(* IEC 61131-3 sources: SmartHomeNew/snapshots/2026-05-25 (part 4) *)

(* ---- FB_Water_Output_Reconciliation.st ---- *)
FUNCTION_BLOCK FB_Water_Output_Reconciliation
VAR_INPUT
    VI_Enable : BOOL;
    VI_System_Time_MS : UDINT;
END_VAR
VAR
    L_i : INT;
    L_Output : ST_Water_Output_Projection_State;
    L_Valve : ST_Water_Valve_Runtime_State;
    L_State : ST_Water_Output_Reconciliation_State;
    L_Any_Runtime_Mismatch : BOOL;
    L_Any_Confirmation_Mismatch : BOOL;
    L_Any_Conflict : BOOL;
END_VAR

IF NOT VI_Enable THEN
    GVL_Water_Output_Reconciliation.G_Runtime_Valid := FALSE;
    RETURN;
END_IF;

L_Any_Runtime_Mismatch := FALSE;
L_Any_Confirmation_Mismatch := FALSE;
L_Any_Conflict := FALSE;

FOR L_i := 1 TO GVL_CONSTANTS.C_MAX_FLOOD_SENSORS DO

    L_Output := GVL_Water_Output_Projection.G_Output_Projection_State[L_i];
    L_Valve := GVL_Water_Valve_Runtime.G_Valve_Runtime_State[L_i];

    // Reset all reconciliation fields per sensor to prevent state leakage across loop iterations.
    L_State.Runtime_Valid := FALSE;
    L_State.Runtime_System_Time_MS := 0;
    L_State.Valve_Group_Id := 0;
    L_State.Projection_Active := FALSE;
    L_State.Runtime_Output_Active := FALSE;
    L_State.Expected_Closed := FALSE;
    L_State.Confirmed_Closed := FALSE;
    L_State.Confirmation_Unknown := FALSE;
    L_State.Reconciliation_Healthy := FALSE;
    L_State.Projection_Runtime_Mismatch := FALSE;
    L_State.Projection_Confirmation_Mismatch := FALSE;
    L_State.Conflict_Detected := FALSE;
    L_State.Topology_Invalid := FALSE;
    L_State.Status_Code := 0;
    L_State.Status_Text := '';

    L_State.Runtime_Valid := TRUE;
    L_State.Runtime_System_Time_MS := VI_System_Time_MS;

    L_State.Valve_Group_Id := L_Output.Valve_Group_Id;
    L_State.Projection_Active := L_Output.Physical_Close_Project;
    L_State.Runtime_Output_Active := L_Valve.Physical_Output_Active;
    L_State.Expected_Closed := L_Output.Expected_Closed;
    L_State.Confirmed_Closed := L_Valve.Confirmed_Closed;
    L_State.Confirmation_Unknown := L_Valve.Confirmation_Unknown;

    IF L_Valve.Confirmation_Available THEN

        IF L_State.Projection_Active <> L_State.Runtime_Output_Active THEN
            L_State.Projection_Runtime_Mismatch := TRUE;
        END_IF;

        IF L_State.Expected_Closed
           AND NOT L_State.Confirmed_Closed THEN
            L_State.Projection_Confirmation_Mismatch := TRUE;
        END_IF;

    END_IF;

    IF L_Output.Projection_Allowed
       AND L_Output.Projection_Denied THEN
        L_State.Conflict_Detected := TRUE;
    END_IF;

    IF L_Output.Valve_Group_Id = 0 THEN
        L_State.Topology_Invalid := TRUE;
    END_IF;

    L_State.Reconciliation_Healthy :=
        NOT L_State.Projection_Runtime_Mismatch
        AND NOT L_State.Projection_Confirmation_Mismatch
        AND NOT L_State.Conflict_Detected
        AND NOT L_State.Topology_Invalid;

    IF L_State.Conflict_Detected THEN
        L_State.Status_Code := 3;
        L_State.Status_Text := 'Projection conflict detected';
    ELSIF L_State.Projection_Runtime_Mismatch THEN
        L_State.Status_Code := 2;
        L_State.Status_Text := 'Projection runtime mismatch';
        L_Any_Runtime_Mismatch := TRUE;
    ELSIF L_State.Projection_Confirmation_Mismatch THEN
        L_State.Status_Code := 1;
        L_State.Status_Text := 'Projection confirmation mismatch';
        L_Any_Confirmation_Mismatch := TRUE;
    ELSE
        L_State.Status_Code := 0;
        L_State.Status_Text := 'Reconciliation healthy';
    END_IF;

    IF L_State.Conflict_Detected THEN
        L_Any_Conflict := TRUE;
    END_IF;

    GVL_Water_Output_Reconciliation.G_Reconciliation_State[L_i] := L_State;
END_FOR;

GVL_Water_Output_Reconciliation.G_Any_Runtime_Mismatch := L_Any_Runtime_Mismatch;
GVL_Water_Output_Reconciliation.G_Any_Confirmation_Mismatch := L_Any_Confirmation_Mismatch;
GVL_Water_Output_Reconciliation.G_Any_Conflict_Detected := L_Any_Conflict;
GVL_Water_Output_Reconciliation.G_Runtime_Valid := TRUE;
GVL_Water_Output_Reconciliation.G_Last_Update_MS := VI_System_Time_MS;

IF L_Any_Conflict THEN
    GVL_Water_Output_Reconciliation.G_Status_Code := 3;
    GVL_Water_Output_Reconciliation.G_Status_Text := 'Water output reconciliation conflict';
ELSIF L_Any_Runtime_Mismatch THEN
    GVL_Water_Output_Reconciliation.G_Status_Code := 2;
    GVL_Water_Output_Reconciliation.G_Status_Text := 'Water output runtime mismatch';
ELSIF L_Any_Confirmation_Mismatch THEN
    GVL_Water_Output_Reconciliation.G_Status_Code := 1;
    GVL_Water_Output_Reconciliation.G_Status_Text := 'Water output confirmation mismatch';
ELSE
    GVL_Water_Output_Reconciliation.G_Status_Code := 0;
    GVL_Water_Output_Reconciliation.G_Status_Text := 'Water output reconciliation healthy';
END_IF;

END_FUNCTION_BLOCK

(* ---- MAIN.st ---- *)
PROGRAM MAIN
// ==============================================================================
// MAIN — deterministic PLC scan-cycle phase map.
// ==============================================================================
// Execution order is preserved by PRG_Main_Phase_* programs.
// No phase gating or controlled shedding is applied here yet.
// Compile/runtime validation must confirm that all referenced phase programs are
// linked by the PLC project export.
// ==============================================================================

PRG_Main_Phase_01_Bootstrap();
PRG_Main_Phase_02_Redundancy();
PRG_Main_Phase_03_Input_Safety_Command();
PRG_Main_Phase_04_Transport_Distributed();
PRG_Main_Phase_05_Domain_Output();
PRG_Main_Phase_06_PostOutput_Authority();
PRG_Main_Phase_07_Semantic_Governance();
PRG_Main_Phase_08_Diagnostics_HMI();

// >>> BULK_SYNC_ANCHOR: MAIN <<<
END_PROGRAM

(* ---- PRG_Access.st ---- *)
PROGRAM PRG_Access
VAR
    fbProjection : FB_Access_Output_Projection;

    fbPulseLock1Open : FB_Access_Pulse_Channel;
    fbPulseLock1Close : FB_Access_Pulse_Channel;
    fbPulseLock2Open : FB_Access_Pulse_Channel;
    fbPulseLock2Close : FB_Access_Pulse_Channel;
    fbPulseGateOpen : FB_Access_Pulse_Channel;
    fbPulseWicketOpen : FB_Access_Pulse_Channel;

    L_Mode : E_Safety_Mode;
    L_Now_MS : UDINT;
    L_Pulse_MS : UDINT;

    L_Distributed_Execute_Allowed : BOOL;
    L_Distributed_Access_Allowed : BOOL;

    L_Lock_1_Open : BOOL;
    L_Lock_1_Close : BOOL;
    L_Lock_2_Open : BOOL;
    L_Lock_2_Close : BOOL;
    L_Gate_Open : BOOL;
    L_Wicket_Open : BOOL;
END_VAR

L_Mode := GVL_SAFETY_SHUTDOWN.G_Safety_Mode;
L_Now_MS := GVL_STATUS.G_System_Time_MS;

GVL_ACCESS_RUNTIME.G_Runtime_Required := FALSE;
GVL_ACCESS_RUNTIME.G_Runtime_Executed := TRUE;
GVL_ACCESS_RUNTIME.G_Runtime_Idle_By_Design := FALSE;
GVL_ACCESS_RUNTIME.G_Runtime_Blocked_By_Distributed_Gates := FALSE;
GVL_ACCESS_RUNTIME.G_Any_Pulse_Active := FALSE;
GVL_ACCESS_RUNTIME.G_Last_Update_MS := L_Now_MS;

// Distributed runtime governance.
// FIRE/GAS emergency semantics remain authoritative.
L_Distributed_Execute_Allowed :=
    GVL_Distributed_Execution_Gates.G_Can_Execute;

L_Distributed_Access_Allowed :=
    GVL_Distributed_Execution_Gates.G_Can_Own_Projection;

IF (L_Mode <> FIRE)
   AND (L_Mode <> GAS)
   AND (
        NOT L_Distributed_Execute_Allowed
        OR NOT L_Distributed_Access_Allowed
       ) THEN

    // Clear all pulse channels before blocking projection to avoid stale pulse-active state.
    fbPulseLock1Open(VI_Command := FALSE, VI_Reset := TRUE, VI_Now_MS := L_Now_MS, VI_Pulse_MS := 100);
    fbPulseLock1Close(VI_Command := FALSE, VI_Reset := TRUE, VI_Now_MS := L_Now_MS, VI_Pulse_MS := 100);
    fbPulseLock2Open(VI_Command := FALSE, VI_Reset := TRUE, VI_Now_MS := L_Now_MS, VI_Pulse_MS := 100);
    fbPulseLock2Close(VI_Command := FALSE, VI_Reset := TRUE, VI_Now_MS := L_Now_MS, VI_Pulse_MS := 100);
    fbPulseGateOpen(VI_Command := FALSE, VI_Reset := TRUE, VI_Now_MS := L_Now_MS, VI_Pulse_MS := 100);
    fbPulseWicketOpen(VI_Command := FALSE, VI_Reset := TRUE, VI_Now_MS := L_Now_MS, VI_Pulse_MS := 100);

    fbProjection(
        VI_Lock_1_Open := FALSE,
        VI_Lock_1_Close := FALSE,
        VI_Lock_2_Open := FALSE,
        VI_Lock_2_Close := FALSE,
        VI_Gate_Open := FALSE,
        VI_Wicket_Open := FALSE
    );

    GVL_ACCESS_RUNTIME.G_Runtime_Blocked_By_Distributed_Gates := TRUE;
    GVL_ACCESS_RUNTIME.G_Any_Pulse_Active := FALSE;
    GVL_ACCESS_RUNTIME.G_Status_Code := 2;
    GVL_ACCESS_RUNTIME.G_Status_Text := 'Access runtime blocked by distributed gates';

    RETURN;
END_IF;

// Load pulse duration from config with safety clamp.
L_Pulse_MS := GVL_CONFIG.G_Access_Pulse_MS;
IF L_Pulse_MS < 100 THEN
    L_Pulse_MS := 100;
ELSIF L_Pulse_MS > 5000 THEN
    L_Pulse_MS := 5000;
END_IF;

L_Lock_1_Open := FALSE;
L_Lock_1_Close := FALSE;
L_Lock_2_Open := FALSE;
L_Lock_2_Close := FALSE;
L_Gate_Open := FALSE;
L_Wicket_Open := FALSE;

CASE L_Mode OF
    FIRE:
        // Fire evacuation access commands are authoritative and continuous.
        L_Lock_1_Open := GVL_COMMAND_SHADOW.G_Lock_1_Open;
        L_Lock_2_Open := GVL_COMMAND_SHADOW.G_Lock_2_Open;
        L_Gate_Open := GVL_COMMAND_SHADOW.G_Gate_Open;
        L_Wicket_Open := GVL_COMMAND_SHADOW.G_Wicket_Open;

        // Synchronize pulse channels with current command state and clear active pulses.
        fbPulseLock1Open(VI_Command := GVL_COMMAND_SHADOW.G_Lock_1_Open, VI_Reset := TRUE, VI_Now_MS := L_Now_MS, VI_Pulse_MS := L_Pulse_MS);
        fbPulseLock1Close(VI_Command := GVL_COMMAND_SHADOW.G_Lock_1_Close, VI_Reset := TRUE, VI_Now_MS := L_Now_MS, VI_Pulse_MS := L_Pulse_MS);
        fbPulseLock2Open(VI_Command := GVL_COMMAND_SHADOW.G_Lock_2_Open, VI_Reset := TRUE, VI_Now_MS := L_Now_MS, VI_Pulse_MS := L_Pulse_MS);
        fbPulseLock2Close(VI_Command := GVL_COMMAND_SHADOW.G_Lock_2_Close, VI_Reset := TRUE, VI_Now_MS := L_Now_MS, VI_Pulse_MS := L_Pulse_MS);
        fbPulseGateOpen(VI_Command := GVL_COMMAND_SHADOW.G_Gate_Open, VI_Reset := TRUE, VI_Now_MS := L_Now_MS, VI_Pulse_MS := L_Pulse_MS);
        fbPulseWicketOpen(VI_Command := GVL_COMMAND_SHADOW.G_Wicket_Open, VI_Reset := TRUE, VI_Now_MS := L_Now_MS, VI_Pulse_MS := L_Pulse_MS);

    GAS:
        // Gas mode uses direct gate opening plus limited pulsed pedestrian/lock release.
        L_Gate_Open := GVL_COMMAND_SHADOW.G_Gate_Open;

        fbPulseLock1Open(VI_Command := GVL_COMMAND_SHADOW.G_Lock_1_Open, VI_Reset := FALSE, VI_Now_MS := L_Now_MS, VI_Pulse_MS := L_Pulse_MS);
        fbPulseLock2Open(VI_Command := GVL_COMMAND_SHADOW.G_Lock_2_Open, VI_Reset := FALSE, VI_Now_MS := L_Now_MS, VI_Pulse_MS := L_Pulse_MS);
        fbPulseWicketOpen(VI_Command := GVL_COMMAND_SHADOW.G_Wicket_Open, VI_Reset := FALSE, VI_Now_MS := L_Now_MS, VI_Pulse_MS := L_Pulse_MS);

        fbPulseLock1Close(VI_Command := GVL_COMMAND_SHADOW.G_Lock_1_Close, VI_Reset := TRUE, VI_Now_MS := L_Now_MS, VI_Pulse_MS := L_Pulse_MS);
        fbPulseLock2Close(VI_Command := GVL_COMMAND_SHADOW.G_Lock_2_Close, VI_Reset := TRUE, VI_Now_MS := L_Now_MS, VI_Pulse_MS := L_Pulse_MS);
        fbPulseGateOpen(VI_Command := GVL_COMMAND_SHADOW.G_Gate_Open, VI_Reset := TRUE, VI_Now_MS := L_Now_MS, VI_Pulse_MS := L_Pulse_MS);

        L_Lock_1_Open := fbPulseLock1Open.VO_Output;
        L_Lock_2_Open := fbPulseLock2Open.VO_Output;
        L_Wicket_Open := fbPulseWicketOpen.VO_Output;

ELSE
        fbPulseLock1Open(VI_Command := GVL_COMMAND_SHADOW.G_Lock_1_Open, VI_Reset := FALSE, VI_Now_MS := L_Now_MS, VI_Pulse_MS := L_Pulse_MS);
        fbPulseLock1Close(VI_Command := GVL_COMMAND_SHADOW.G_Lock_1_Close, VI_Reset := FALSE, VI_Now_MS := L_Now_MS, VI_Pulse_MS := L_Pulse_MS);
        fbPulseLock2Open(VI_Command := GVL_COMMAND_SHADOW.G_Lock_2_Open, VI_Reset := FALSE, VI_Now_MS := L_Now_MS, VI_Pulse_MS := L_Pulse_MS);
        fbPulseLock2Close(VI_Command := GVL_COMMAND_SHADOW.G_Lock_2_Close, VI_Reset := FALSE, VI_Now_MS := L_Now_MS, VI_Pulse_MS := L_Pulse_MS);
        fbPulseGateOpen(VI_Command := GVL_COMMAND_SHADOW.G_Gate_Open, VI_Reset := FALSE, VI_Now_MS := L_Now_MS, VI_Pulse_MS := L_Pulse_MS);
        fbPulseWicketOpen(VI_Command := GVL_COMMAND_SHADOW.G_Wicket_Open, VI_Reset := FALSE, VI_Now_MS := L_Now_MS, VI_Pulse_MS := L_Pulse_MS);

        L_Lock_1_Open := fbPulseLock1Open.VO_Output;
        L_Lock_1_Close := fbPulseLock1Close.VO_Output;
        L_Lock_2_Open := fbPulseLock2Open.VO_Output;
        L_Lock_2_Close := fbPulseLock2Close.VO_Output;
        L_Gate_Open := fbPulseGateOpen.VO_Output;
        L_Wicket_Open := fbPulseWicketOpen.VO_Output;
END_CASE;

GVL_ACCESS_RUNTIME.G_Any_Pulse_Active :=
    fbPulseLock1Open.VO_Active
    OR fbPulseLock1Close.VO_Active
    OR fbPulseLock2Open.VO_Active
    OR fbPulseLock2Close.VO_Active
    OR fbPulseGateOpen.VO_Active
    OR fbPulseWicketOpen.VO_Active;

GVL_ACCESS_RUNTIME.G_Runtime_Required :=
    (L_Mode = FIRE)
    OR (L_Mode = GAS)
    OR GVL_COMMAND_SHADOW.G_Lock_1_Open
    OR GVL_COMMAND_SHADOW.G_Lock_1_Close
    OR GVL_COMMAND_SHADOW.G_Lock_2_Open
    OR GVL_COMMAND_SHADOW.G_Lock_2_Close
    OR GVL_COMMAND_SHADOW.G_Gate_Open
    OR GVL_COMMAND_SHADOW.G_Wicket_Open
    OR GVL_ACCESS_RUNTIME.G_Any_Pulse_Active;

GVL_ACCESS_RUNTIME.G_Runtime_Idle_By_Design :=
    NOT GVL_ACCESS_RUNTIME.G_Runtime_Required;

IF GVL_ACCESS_RUNTIME.G_Runtime_Idle_By_Design THEN
    GVL_ACCESS_RUNTIME.G_Status_Code := 0;
    GVL_ACCESS_RUNTIME.G_Status_Text := 'Access runtime idle by design';
ELSE
    GVL_ACCESS_RUNTIME.G_Status_Code := 1;
    GVL_ACCESS_RUNTIME.G_Status_Text := 'Access runtime active';
END_IF;

fbProjection(
    VI_Lock_1_Open := L_Lock_1_Open,
    VI_Lock_1_Close := L_Lock_1_Close,
    VI_Lock_2_Open := L_Lock_2_Open,
    VI_Lock_2_Close := L_Lock_2_Close,
    VI_Gate_Open := L_Gate_Open,
    VI_Wicket_Open := L_Wicket_Open
);

// >>> BULK_SYNC_ANCHOR: PRG_Access <<<
END_PROGRAM

(* ---- PRG_Authority_Lineage_Governor.st ---- *)
PROGRAM PRG_Authority_Lineage_Governor
VAR
    L_Now_MS : UDINT;
    L_Lineage_Valid : BOOL := TRUE;
    L_Error_Code : UDINT := 0;
    L_Error_Text : STRING(160) := '';
END_VAR

L_Now_MS := GVL_STATUS.G_System_Time_MS;
L_Lineage_Valid := TRUE;
L_Error_Code := 0;
L_Error_Text := '';

GVL_AUTHORITY_LINEAGE.Authority_Lineage_Valid := FALSE;
GVL_AUTHORITY_LINEAGE.Warm_Restart_Continuity_Valid := FALSE;
GVL_AUTHORITY_LINEAGE.HA_Resume_Continuity_Valid := FALSE;
GVL_AUTHORITY_LINEAGE.Retained_State_Integrity_Valid := FALSE;

IF GVL_AUTHORITY_LINEAGE.Authority_Replay_Suspected THEN
    L_Lineage_Valid := FALSE;
    L_Error_Code := 25000;
    L_Error_Text := 'Authority replay suspected';
END_IF;

IF L_Lineage_Valid AND GVL_AUTHORITY_LINEAGE.Retained_State_Skew_Detected THEN
    L_Lineage_Valid := FALSE;
    L_Error_Code := 25001;
    L_Error_Text := 'Retained state skew detected';
END_IF;

IF L_Lineage_Valid AND GVL_AUTHORITY_LINEAGE.Partial_Authority_Resurrection_Detected THEN
    L_Lineage_Valid := FALSE;
    L_Error_Code := 25002;
    L_Error_Text := 'Partial authority resurrection detected';
END_IF;

IF L_Lineage_Valid AND GVL_AUTHORITY_LINEAGE.Epoch_Lineage_Discontinuity_Detected THEN
    L_Lineage_Valid := FALSE;
    L_Error_Code := 25003;
    L_Error_Text := 'Epoch lineage discontinuity detected';
END_IF;

IF L_Lineage_Valid
AND (ULINT_TO_UDINT(GVL_PHYSICAL_AUTHORITY_EPOCH.Physical_Authority_Epoch) < GVL_AUTHORITY_LINEAGE.Last_Physical_Authority_Epoch) THEN
    GVL_AUTHORITY_LINEAGE.Authority_Replay_Suspected := TRUE;
    L_Lineage_Valid := FALSE;
    L_Error_Code := 25010;
    L_Error_Text := 'Physical authority epoch rollback detected';
END_IF;

IF L_Lineage_Valid
AND (ULINT_TO_UDINT(GVL_RUNTIME_EPOCH.Runtime_Epoch) < GVL_AUTHORITY_LINEAGE.Last_Runtime_Epoch) THEN
    GVL_AUTHORITY_LINEAGE.Retained_State_Skew_Detected := TRUE;
    L_Lineage_Valid := FALSE;
    L_Error_Code := 25011;
    L_Error_Text := 'Runtime epoch rollback detected';
END_IF;

IF L_Lineage_Valid
AND (ULINT_TO_UDINT(GVL_OUTPUT_EPOCH.Output_Publication_Epoch) < GVL_AUTHORITY_LINEAGE.Last_Output_Publication_Epoch) THEN
    GVL_AUTHORITY_LINEAGE.Partial_Authority_Resurrection_Detected := TRUE;
    L_Lineage_Valid := FALSE;
    L_Error_Code := 25012;
    L_Error_Text := 'Output publication epoch rollback detected';
END_IF;

IF L_Lineage_Valid THEN
    GVL_AUTHORITY_LINEAGE.Authority_Lineage_Valid := TRUE;
    GVL_AUTHORITY_LINEAGE.Warm_Restart_Continuity_Valid := TRUE;
    GVL_AUTHORITY_LINEAGE.HA_Resume_Continuity_Valid := TRUE;
    GVL_AUTHORITY_LINEAGE.Retained_State_Integrity_Valid := TRUE;

    GVL_AUTHORITY_LINEAGE.Authority_Lineage_Epoch := ULINT_TO_UDINT(GVL_PHYSICAL_AUTHORITY_EPOCH.Physical_Authority_Epoch);
    GVL_AUTHORITY_LINEAGE.Last_Physical_Authority_Epoch := ULINT_TO_UDINT(GVL_PHYSICAL_AUTHORITY_EPOCH.Physical_Authority_Epoch);
    GVL_AUTHORITY_LINEAGE.Last_Runtime_Epoch := ULINT_TO_UDINT(GVL_RUNTIME_EPOCH.Runtime_Epoch);
    GVL_AUTHORITY_LINEAGE.Last_Output_Publication_Epoch := ULINT_TO_UDINT(GVL_OUTPUT_EPOCH.Output_Publication_Epoch);
    GVL_AUTHORITY_LINEAGE.Authority_Lineage_Last_Update_MS := L_Now_MS;
    GVL_AUTHORITY_LINEAGE.Authority_Lineage_Last_Error_Code := 0;
    GVL_AUTHORITY_LINEAGE.Authority_Lineage_Last_Error_Text := '';
ELSE
    GVL_AUTHORITY_LINEAGE.Authority_Lineage_Valid := FALSE;
    GVL_AUTHORITY_LINEAGE.Authority_Lineage_Last_Error_Code := L_Error_Code;
    GVL_AUTHORITY_LINEAGE.Authority_Lineage_Last_Error_Text := L_Error_Text;
    GVL_AUTHORITY_LINEAGE.Authority_Lineage_Invalidation_Count := GVL_AUTHORITY_LINEAGE.Authority_Lineage_Invalidation_Count + 1;
END_IF;

END_PROGRAM

(* ---- PRG_Authority_Restoration_Governor.st ---- *)
PROGRAM PRG_Authority_Restoration_Governor
VAR
    L_Now_MS : UDINT;
    L_Restoration_Valid : BOOL := TRUE;
END_VAR

L_Now_MS := GVL_STATUS.G_System_Time_MS;
L_Restoration_Valid := TRUE;

GVL_AUTHORITY_RESTORATION.Authority_Restoration_Active := FALSE;
GVL_AUTHORITY_RESTORATION.Authority_Restoration_Allowed := FALSE;
GVL_AUTHORITY_RESTORATION.Authority_Restoration_Completed := FALSE;

GVL_AUTHORITY_RESTORATION.Snapshot_Restoration_Valid := FALSE;
GVL_AUTHORITY_RESTORATION.Consensus_Restoration_Valid := FALSE;
GVL_AUTHORITY_RESTORATION.Causality_Restoration_Valid := FALSE;
GVL_AUTHORITY_RESTORATION.Epoch_Restoration_Valid := FALSE;
GVL_AUTHORITY_RESTORATION.Lineage_Restoration_Valid := FALSE;

GVL_AUTHORITY_RESTORATION.Revocation_Clearance_Valid := FALSE;
GVL_AUTHORITY_RESTORATION.Stabilization_Window_Elapsed := FALSE;
GVL_AUTHORITY_RESTORATION.Reauthorization_Order_Valid := FALSE;

IF GVL_AUTHORITY_REVOCATION.Authority_Revocation_Active THEN
    L_Restoration_Valid := FALSE;
END_IF;

IF L_Restoration_Valid
AND (
    GVL_SAFETY_SHUTDOWN.G_Safety_Active
    OR GVL_SAFETY_RECOVERY.G_Recovery_Active
    OR (GVL_SAFETY_RECOVERY.G_Recovery_Phase <> IDLE)
) THEN
    L_Restoration_Valid := FALSE;
END_IF;

IF L_Restoration_Valid
AND NOT GVL_PHYSICAL_SNAPSHOT.Physical_Snapshot_Valid THEN
    L_Restoration_Valid := FALSE;
END_IF;

IF L_Restoration_Valid THEN
    GVL_AUTHORITY_RESTORATION.Snapshot_Restoration_Valid := TRUE;
END_IF;

IF L_Restoration_Valid
AND NOT GVL_SENSOR_CONSENSUS.Sensor_Consensus_Valid THEN
    L_Restoration_Valid := FALSE;
END_IF;

IF L_Restoration_Valid THEN
    GVL_AUTHORITY_RESTORATION.Consensus_Restoration_Valid := TRUE;
END_IF;

IF L_Restoration_Valid
AND NOT GVL_TELEMETRY.Command_Telemetry_Causality_Valid THEN
    L_Restoration_Valid := FALSE;
END_IF;

IF L_Restoration_Valid THEN
    GVL_AUTHORITY_RESTORATION.Causality_Restoration_Valid := TRUE;
END_IF;

IF L_Restoration_Valid
AND NOT GVL_PHYSICAL_AUTHORITY_EPOCH.Physical_Authority_Epoch_Valid THEN
    L_Restoration_Valid := FALSE;
END_IF;

IF L_Restoration_Valid THEN
    GVL_AUTHORITY_RESTORATION.Epoch_Restoration_Valid := TRUE;
END_IF;

IF L_Restoration_Valid
AND NOT GVL_AUTHORITY_LINEAGE.Authority_Lineage_Valid THEN
    L_Restoration_Valid := FALSE;
END_IF;

IF L_Restoration_Valid THEN
    GVL_AUTHORITY_RESTORATION.Lineage_Restoration_Valid := TRUE;
END_IF;

IF L_Restoration_Valid
AND GVL_AUTHORITY_REVOCATION.Quarantine_Fabric_Active THEN
    L_Restoration_Valid := FALSE;
END_IF;

IF L_Restoration_Valid THEN
    GVL_AUTHORITY_RESTORATION.Revocation_Clearance_Valid := TRUE;
END_IF;

IF L_Restoration_Valid
AND ((L_Now_MS - GVL_AUTHORITY_REVOCATION.Revocation_Last_Update_MS) < 5000) THEN
    L_Restoration_Valid := FALSE;
END_IF;

IF L_Restoration_Valid THEN
    GVL_AUTHORITY_RESTORATION.Stabilization_Window_Elapsed := TRUE;
END_IF;

IF L_Restoration_Valid THEN
    GVL_AUTHORITY_RESTORATION.Authority_Restoration_Active := TRUE;
    GVL_AUTHORITY_RESTORATION.Authority_Restoration_Allowed := TRUE;
    GVL_AUTHORITY_RESTORATION.Authority_Restoration_Completed := TRUE;
    GVL_AUTHORITY_RESTORATION.Reauthorization_Order_Valid := TRUE;
    GVL_AUTHORITY_RESTORATION.Restoration_Epoch :=
        GVL_PHYSICAL_AUTHORITY_EPOCH.Physical_Authority_Epoch;
    GVL_AUTHORITY_RESTORATION.Restoration_Last_Update_MS := L_Now_MS;
END_IF;

END_PROGRAM

(* ---- PRG_Away_Restore_Manager.st ---- *)
PROGRAM PRG_Away_Restore_Manager
VAR
    L_i : INT;
    L_Away_Active_Prev : BOOL := FALSE;
    L_Away_Level_Prev : BYTE := 0;
    L_Take_Snapshot : BOOL;
    L_Start_Restore : BOOL;
END_VAR

// Complete cleanup one cycle after publishing progress=1.0. This lets domain
// output managers consume the final restore state before snapshot invalidation.
IF GVL_AWAY_RESTORE.G_Restore_Finalize_Pending THEN
    GVL_AWAY_RESTORE.G_Restore_Active := FALSE;
    GVL_AWAY_RESTORE.G_Restore_Done := TRUE;
    GVL_AWAY_RESTORE.G_Snapshot_Valid := FALSE;
    GVL_AWAY_RESTORE.G_Restore_Finalize_Pending := FALSE;
    GVL_AWAY_RESTORE.G_Restore_Progress := 0.0;
END_IF;

L_Take_Snapshot :=
    GVL_POLICY.G_Away_Active AND
    (GVL_POLICY.G_Away_Level = 1) AND
    (NOT L_Away_Active_Prev);

IF L_Take_Snapshot THEN
    FOR L_i := 1 TO GVL_CONSTANTS.C_MAX_LIGHT_ZONES DO
        GVL_AWAY_RESTORE.G_Lighting_Levels[L_i] := GVL_STATE.G_Lighting_Levels[L_i];
    END_FOR;

    FOR L_i := 1 TO GVL_CONSTANTS.C_MAX_SOCKETS DO
        GVL_AWAY_RESTORE.G_Socket_States[L_i] := GVL_STATE.G_Socket_States[L_i];
    END_FOR;

    GVL_AWAY_RESTORE.G_Snapshot_Valid := TRUE;
    GVL_AWAY_RESTORE.G_Snapshot_Taken_MS := GVL_TIME_SERVICE.G_Now_MS;
    GVL_AWAY_RESTORE.G_Restore_Done := FALSE;
    GVL_AWAY_RESTORE.G_Restore_Finalize_Pending := FALSE;
END_IF;

L_Start_Restore :=
    GVL_POLICY.G_Away_Restore_Requested AND
    GVL_AWAY_RESTORE.G_Snapshot_Valid;

IF L_Start_Restore THEN
    GVL_AWAY_RESTORE.G_Restore_Active := TRUE;
    GVL_AWAY_RESTORE.G_Restore_Started_MS := GVL_TIME_SERVICE.G_Now_MS;
    GVL_AWAY_RESTORE.G_Restore_Done := FALSE;
    GVL_AWAY_RESTORE.G_Restore_Finalize_Pending := FALSE;
END_IF;

IF GVL_AWAY_RESTORE.G_Restore_Active THEN
    GVL_AWAY_RESTORE.G_Restore_Progress := GVL_POLICY.G_Away_Restore_Progress;

    IF NOT GVL_POLICY.G_Away_Restore_Active THEN
        GVL_AWAY_RESTORE.G_Restore_Progress := 1.0;
        GVL_AWAY_RESTORE.G_Restore_Finalize_Pending := TRUE;
    END_IF;
ELSE
    IF NOT GVL_AWAY_RESTORE.G_Restore_Done THEN
        GVL_AWAY_RESTORE.G_Restore_Progress := 0.0;
    END_IF;
END_IF;

L_Away_Active_Prev := GVL_POLICY.G_Away_Active;
L_Away_Level_Prev := GVL_POLICY.G_Away_Level;

END_PROGRAM

(* ---- PRG_Causal_Narrative_Engine.st ---- *)
PROGRAM PRG_Causal_Narrative_Engine
// PASSIVE CAUSAL NARRATIVE ENGINE
// HUMAN-READABLE SEMANTIC PROJECTION

GVL_CAUSAL_NARRATIVE_FABRIC.Narrative_Causality_Coherent :=
    GVL_TEMPORAL_CAUSALITY_CLOSURE_FABRIC.Temporal_Causality_Coherent;

GVL_CAUSAL_NARRATIVE_FABRIC.Narrative_Runtime_Alignment_Valid :=
    GVL_RUNTIME_TRANSITION_SYSTEM.Runtime_Transition_Legal;

IF GVL_RUNTIME_TRANSITION_SYSTEM.Illegal_Runtime_Transition_Observed THEN
    GVL_CAUSAL_NARRATIVE_FABRIC.Runtime_Narrative_Available := TRUE;
    GVL_CAUSAL_NARRATIVE_FABRIC.Runtime_Narrative_Code :=
        'transition legality violation observed';
END_IF;

IF GVL_RUNTIME_TRANSITION_SYSTEM.Recovery_Without_Lineage_Observed THEN
    GVL_CAUSAL_NARRATIVE_FABRIC.Recovery_Narrative_Available := TRUE;
    GVL_CAUSAL_NARRATIVE_FABRIC.Recovery_Narrative_Code :=
        'recovery blocked by lineage instability';
END_IF;

IF GVL_RUNTIME_TRANSITION_SYSTEM.Unsafe_Trust_Escalation_Observed THEN
    GVL_CAUSAL_NARRATIVE_FABRIC.Authority_Narrative_Available := TRUE;
    GVL_CAUSAL_NARRATIVE_FABRIC.Authority_Narrative_Code :=
        'unsafe trust escalation detected';
END_IF;

END_PROGRAM

(* ---- PRG_Causality_Reversal_Prevention_Governor.st ---- *)
PROGRAM PRG_Causality_Reversal_Prevention_Governor
IF GVL_HISTORICAL_ORDERING_INTEGRITY_FABRIC.Historical_Ordering_Integrity_Granted
AND NOT GVL_CAUSALITY_REVERSAL_PREVENTION_FABRIC.Causality_Reversal_Detected
AND NOT GVL_CAUSALITY_REVERSAL_PREVENTION_FABRIC.Resurrection_After_Revocation_Detected
AND NOT GVL_CAUSALITY_REVERSAL_PREVENTION_FABRIC.Unsafe_Temporal_Replay_Detected THEN

    GVL_CAUSALITY_REVERSAL_PREVENTION_FABRIC.Causality_Reversal_Prevention_Valid := TRUE;
    GVL_CAUSALITY_REVERSAL_PREVENTION_FABRIC.Causality_Reversal_Prevention_Granted := TRUE;
    GVL_CAUSALITY_REVERSAL_PREVENTION_FABRIC.Causality_Reversal_Prevented := TRUE;
    GVL_CAUSALITY_REVERSAL_PREVENTION_FABRIC.Authority_Ordering_Canonical := TRUE;
    GVL_CAUSALITY_REVERSAL_PREVENTION_FABRIC.Revocation_Resurrection_Boundary_Stable := TRUE;
END_IF;
END_PROGRAM

(* ---- PRG_Command_Arbitration_Phase_01_Reset_Role.st ---- *)
PROGRAM PRG_Command_Arbitration_Phase_01_Reset_Role
// Command arbitration phase 01: reset deterministic buffer and handle PLC role gates.
// Preserves old priority 1/2 early-exit semantics through buffer flags.

GVL_COMMAND_ARBITRATION_BUFFER.B_Mode := GVL_SAFETY_SHUTDOWN.G_Safety_Mode;
GVL_COMMAND_ARBITRATION_BUFFER.B_Safety_Active := FALSE;
GVL_COMMAND_ARBITRATION_BUFFER.B_User_Access_OK := FALSE;
GVL_COMMAND_ARBITRATION_BUFFER.B_Role_Conflict_Active := FALSE;
GVL_COMMAND_ARBITRATION_BUFFER.B_PLC_Inactive_Active := FALSE;

GVL_COMMAND_ARBITRATION_BUFFER.B_Gas_Valve_Close := FALSE;
GVL_COMMAND_ARBITRATION_BUFFER.B_Boiler_Stop := FALSE;
GVL_COMMAND_ARBITRATION_BUFFER.B_Supply_100_Req := FALSE;
GVL_COMMAND_ARBITRATION_BUFFER.B_Supply_80_Req := FALSE;
GVL_COMMAND_ARBITRATION_BUFFER.B_Vent_PV3_Boost := FALSE;
GVL_COMMAND_ARBITRATION_BUFFER.B_Exhaust_100_Req := FALSE;
GVL_COMMAND_ARBITRATION_BUFFER.B_Vent_Stop := FALSE;
GVL_COMMAND_ARBITRATION_BUFFER.B_Vent_Block := FALSE;
GVL_COMMAND_ARBITRATION_BUFFER.B_Vent_Smoke_Exhaust := FALSE;

GVL_COMMAND_ARBITRATION_BUFFER.B_Heating_Block := FALSE;
GVL_COMMAND_ARBITRATION_BUFFER.B_Heating_Emergency_Stop := FALSE;
GVL_COMMAND_ARBITRATION_BUFFER.B_Heating_Gas_Safety_Stop := FALSE;

GVL_COMMAND_ARBITRATION_BUFFER.B_Water_Block := FALSE;
GVL_COMMAND_ARBITRATION_BUFFER.B_Water_Emergency_Stop := FALSE;
GVL_COMMAND_ARBITRATION_BUFFER.B_Close_Valve_35 := FALSE;
GVL_COMMAND_ARBITRATION_BUFFER.B_Close_Valve_36 := FALSE;

GVL_COMMAND_ARBITRATION_BUFFER.B_Lock_1_Open := FALSE;
GVL_COMMAND_ARBITRATION_BUFFER.B_Lock_1_Close := FALSE;
GVL_COMMAND_ARBITRATION_BUFFER.B_Lock_2_Open := FALSE;
GVL_COMMAND_ARBITRATION_BUFFER.B_Lock_2_Close := FALSE;
GVL_COMMAND_ARBITRATION_BUFFER.B_Gate_Open := FALSE;
GVL_COMMAND_ARBITRATION_BUFFER.B_Wicket_Open := FALSE;

IF GVL_STATUS.G_Is_Active_PLC AND GVL_STATUS.G_Other_PLC_Is_Active THEN
    GVL_HEALTH_BRIDGE.G_Role_Conflict_Error := TRUE;
    GVL_COMMAND_ARBITRATION_BUFFER.B_Role_Conflict_Active := TRUE;

    GVL_COMMAND_ARBITRATION_BUFFER.B_Gas_Valve_Close := TRUE;
    GVL_COMMAND_ARBITRATION_BUFFER.B_Boiler_Stop := TRUE;
    GVL_COMMAND_ARBITRATION_BUFFER.B_Vent_Stop := TRUE;
    GVL_COMMAND_ARBITRATION_BUFFER.B_Vent_Block := TRUE;

    GVL_COMMAND_ARBITRATION_BUFFER.B_Heating_Block := TRUE;
    GVL_COMMAND_ARBITRATION_BUFFER.B_Heating_Emergency_Stop := TRUE;
    GVL_COMMAND_ARBITRATION_BUFFER.B_Heating_Gas_Safety_Stop := TRUE;

    GVL_COMMAND_ARBITRATION_BUFFER.B_Water_Block := TRUE;
    GVL_COMMAND_ARBITRATION_BUFFER.B_Water_Emergency_Stop := TRUE;
    GVL_COMMAND_ARBITRATION_BUFFER.B_Close_Valve_35 := TRUE;
    GVL_COMMAND_ARBITRATION_BUFFER.B_Close_Valve_36 := TRUE;

ELSIF NOT GVL_STATUS.G_Is_Active_PLC THEN
    GVL_COMMAND_ARBITRATION_BUFFER.B_PLC_Inactive_Active := TRUE;

    GVL_COMMAND_ARBITRATION_BUFFER.B_Gas_Valve_Close := GVL_COMMAND_POLICY_CONFIG.G_PLC_Inactive_Close_Gas;
    GVL_COMMAND_ARBITRATION_BUFFER.B_Boiler_Stop := GVL_COMMAND_POLICY_CONFIG.G_PLC_Inactive_Stop_Boiler;
    GVL_COMMAND_ARBITRATION_BUFFER.B_Vent_Stop := GVL_COMMAND_POLICY_CONFIG.G_PLC_Inactive_Stop_Vent;
    GVL_COMMAND_ARBITRATION_BUFFER.B_Vent_Block := FALSE;

    GVL_COMMAND_ARBITRATION_BUFFER.B_Heating_Block := GVL_COMMAND_POLICY_CONFIG.G_PLC_Inactive_Block_Heating;
    GVL_COMMAND_ARBITRATION_BUFFER.B_Heating_Emergency_Stop := FALSE;
    GVL_COMMAND_ARBITRATION_BUFFER.B_Heating_Gas_Safety_Stop := FALSE;

    GVL_COMMAND_ARBITRATION_BUFFER.B_Water_Block := GVL_COMMAND_POLICY_CONFIG.G_PLC_Inactive_Block_Water;
    GVL_COMMAND_ARBITRATION_BUFFER.B_Water_Emergency_Stop := FALSE;
    GVL_COMMAND_ARBITRATION_BUFFER.B_Close_Valve_35 := FALSE;
    GVL_COMMAND_ARBITRATION_BUFFER.B_Close_Valve_36 := FALSE;
END_IF;

// >>> BULK_SYNC_ANCHOR: PRG_Command_Arbitration_Phase_01_Reset_Role <<<
END_PROGRAM

(* ---- PRG_Convergence_Governor.st ---- *)
PROGRAM PRG_Convergence_Governor
VAR
    L_Now_MS : UDINT;
    L_Healthy : BOOL := TRUE;
    L_Error_Code : UDINT := 0;
    L_Error_Text : STRING(160) := '';

    L_Recent_Invalidation : BOOL;
    L_Epoch_Advancement_Healthy : BOOL;
END_VAR

L_Now_MS := GVL_STATUS.G_System_Time_MS;
L_Healthy := TRUE;
L_Error_Code := 0;
L_Error_Text := '';

GVL_CONVERGENCE.Convergence_Runtime_Barrier_OK :=
    GVL_RUNTIME_EPOCH.Runtime_Runtime_Barrier_OK
    AND GVL_RUNTIME_EPOCH.Runtime_IO_Publication_Allowed;

GVL_CONVERGENCE.Convergence_Runtime_Snapshot_OK :=
    GVL_RUNTIME_SNAPSHOT.Snapshot_Frozen
    AND GVL_RUNTIME_SNAPSHOT.Snapshot_Publication_Allowed
    AND GVL_RUNTIME_SNAPSHOT.Snapshot_Copy_Valid
    AND GVL_RUNTIME_SNAPSHOT.Snapshot_Isolation_Valid
    AND GVL_RUNTIME_SNAPSHOT.Snapshot_Runtime_Authority_Valid
    AND NOT GVL_RUNTIME_SNAPSHOT.Snapshot_Mutation_Detected;

GVL_CONVERGENCE.Convergence_Distributed_Snapshot_OK :=
    GVL_DISTRIBUTED_SNAPSHOT.Distributed_Publication_Reconciled
    AND GVL_DISTRIBUTED_SNAPSHOT.Distributed_Publication_Freeze_Valid
    AND GVL_DISTRIBUTED_SNAPSHOT.Distributed_Snapshot_Consistent;

GVL_CONVERGENCE.Convergence_Distributed_Commit_OK :=
    GVL_DISTRIBUTED_COMMIT.Distributed_Commit_Valid
    AND GVL_DISTRIBUTED_COMMIT.Publication_Prepare_Valid
    AND GVL_DISTRIBUTED_COMMIT.Publication_Commit_Confirmed
    AND NOT GVL_DISTRIBUTED_COMMIT.Peer_Commit_Mismatch
    AND NOT GVL_DISTRIBUTED_COMMIT.Commit_Lease_Expired;

GVL_CONVERGENCE.Convergence_Semantic_Progress_OK :=
    GVL_SEMANTIC_PROGRESS.Semantic_Forward_Progress_Valid
    AND GVL_SEMANTIC_PROGRESS.Semantic_Execution_Continuity_OK
    AND NOT GVL_SEMANTIC_PROGRESS.Semantic_Stagnation_Detected
    AND NOT GVL_SEMANTIC_PROGRESS.Semantic_Replay_Suspected
    AND NOT GVL_SEMANTIC_PROGRESS.Semantic_Livelock_Suspected
    AND NOT GVL_SEMANTIC_PROGRESS.Semantic_Deadlock_Suspected
    AND NOT GVL_SEMANTIC_PROGRESS.Semantic_Progress_Lease_Expired
    AND NOT GVL_SEMANTIC_PROGRESS.Semantic_Progress_Quarantine_Active;

GVL_CONVERGENCE.Convergence_Output_Freshness_OK :=
    GVL_RUNTIME_EPOCH.Runtime_Runtime_Barrier_OK
    AND GVL_RUNTIME_EPOCH.Runtime_IO_Publication_Allowed
    AND GVL_RUNTIME_SNAPSHOT.Snapshot_Frozen
    AND GVL_RUNTIME_SNAPSHOT.Snapshot_Publication_Allowed
    AND GVL_RUNTIME_SNAPSHOT.Snapshot_Copy_Valid
    AND GVL_RUNTIME_SNAPSHOT.Snapshot_Isolation_Valid
    AND NOT GVL_RUNTIME_SNAPSHOT.Snapshot_Mutation_Detected
    AND GVL_DISTRIBUTED_SNAPSHOT.Distributed_Publication_Reconciled
    AND GVL_DISTRIBUTED_SNAPSHOT.Distributed_Publication_Freeze_Valid
    AND GVL_DISTRIBUTED_SNAPSHOT.Distributed_Snapshot_Consistent
    AND GVL_DISTRIBUTED_COMMIT.Distributed_Commit_Valid
    AND GVL_DISTRIBUTED_COMMIT.Publication_Prepare_Valid
    AND GVL_DISTRIBUTED_COMMIT.Publication_Commit_Confirmed
    AND NOT GVL_DISTRIBUTED_COMMIT.Peer_Commit_Mismatch
    AND NOT GVL_DISTRIBUTED_COMMIT.Commit_Lease_Expired
    AND GVL_OUTPUT_EPOCH.Output_Publication_Valid
    AND GVL_OUTPUT_EPOCH.Output_Runtime_Epoch_Valid
    AND NOT GVL_OUTPUT_EPOCH.Output_Lease_Expired
    AND NOT GVL_OUTPUT_EPOCH.Output_Forced_Safe_Decay
    AND GVL_COMMAND_VERIFY.PreOutput_Barrier_OK
    AND NOT GVL_COMMAND_VERIFY.PreOutput_Block_IO;

// Epoch advancement freshness.
L_Epoch_Advancement_Healthy :=
    (GVL_SEMANTIC_PROGRESS.Semantic_Runtime_Barrier_Epoch -
     GVL_SEMANTIC_PROGRESS.Semantic_Last_Runtime_Barrier_Epoch) <= 2
    AND
    (GVL_SEMANTIC_PROGRESS.Semantic_Distributed_Commit_Epoch -
     GVL_SEMANTIC_PROGRESS.Semantic_Last_Distributed_Commit_Epoch) <= 2
    AND
    (GVL_SEMANTIC_PROGRESS.Semantic_Output_Publication_Epoch -
     GVL_SEMANTIC_PROGRESS.Semantic_Last_Output_Publication_Epoch) <= 2;

// Oscillation damping window.
L_Recent_Invalidation :=
    (L_Now_MS - GVL_CONVERGENCE.Convergence_Last_Invalidation_MS) < 30000;

IF NOT GVL_CONVERGENCE.Convergence_Runtime_Barrier_OK THEN
    L_Healthy := FALSE;
    L_Error_Code := 18000;
    L_Error_Text := 'Runtime barrier convergence invalid';
END_IF;

IF L_Healthy AND NOT GVL_CONVERGENCE.Convergence_Runtime_Snapshot_OK THEN
    L_Healthy := FALSE;
    L_Error_Code := 18001;
    L_Error_Text := 'Runtime snapshot convergence invalid';
END_IF;

IF L_Healthy AND NOT GVL_CONVERGENCE.Convergence_Distributed_Snapshot_OK THEN
    L_Healthy := FALSE;
    L_Error_Code := 18002;
    L_Error_Text := 'Distributed snapshot convergence invalid';
END_IF;

IF L_Healthy AND NOT GVL_CONVERGENCE.Convergence_Distributed_Commit_OK THEN
    L_Healthy := FALSE;
    L_Error_Code := 18003;
    L_Error_Text := 'Distributed commit convergence invalid';
END_IF;

IF L_Healthy AND NOT GVL_CONVERGENCE.Convergence_Semantic_Progress_OK THEN
    L_Healthy := FALSE;
    L_Error_Code := 18004;
    L_Error_Text := 'Semantic progress convergence invalid';
END_IF;

IF L_Healthy AND NOT GVL_CONVERGENCE.Convergence_Output_Freshness_OK THEN
    L_Healthy := FALSE;
    L_Error_Code := 18005;
    L_Error_Text := 'Output freshness convergence invalid';
END_IF;

IF L_Healthy AND NOT L_Epoch_Advancement_Healthy THEN
    L_Healthy := FALSE;
    L_Error_Code := 18006;
    L_Error_Text := 'Epoch advancement freshness invalid';
END_IF;

IF L_Healthy AND L_Recent_Invalidation THEN
    L_Healthy := FALSE;
    L_Error_Code := 18007;
    L_Error_Text := 'Convergence oscillation damping active';
END_IF;

IF L_Healthy THEN
    GVL_CONVERGENCE.Convergence_Healthy_Observed := TRUE;

    GVL_CONVERGENCE.Recovery_Stable_Cycle_Count :=
        GVL_CONVERGENCE.Recovery_Stable_Cycle_Count + 1;

    IF GVL_CONVERGENCE.Convergence_Last_Healthy_MS = 0 THEN
        GVL_CONVERGENCE.Convergence_Last_Healthy_MS := L_Now_MS;
    END_IF;

    GVL_CONVERGENCE.Recovery_Stable_Time_MS :=
        L_Now_MS - GVL_CONVERGENCE.Convergence_Last_Healthy_MS;

    IF (GVL_CONVERGENCE.Recovery_Stable_Cycle_Count >= GVL_CONVERGENCE.Convergence_Min_Stable_Cycles)
    AND (GVL_CONVERGENCE.Recovery_Stable_Time_MS >= GVL_CONVERGENCE.Convergence_Min_Stable_Time_MS)
    THEN
        GVL_CONVERGENCE.Convergence_Lease_OK := TRUE;
        GVL_CONVERGENCE.Convergence_Release_Allowed := TRUE;
    ELSE
        GVL_CONVERGENCE.Convergence_Lease_OK := FALSE;
        GVL_CONVERGENCE.Convergence_Release_Allowed := FALSE;
    END_IF;

    GVL_CONVERGENCE.Convergence_Last_Error_Code := 0;
    GVL_CONVERGENCE.Convergence_Last_Error_Text := '';
ELSE
    GVL_CONVERGENCE.Convergence_Healthy_Observed := FALSE;

    GVL_CONVERGENCE.Recovery_Stable_Cycle_Count := 0;
    GVL_CONVERGENCE.Recovery_Stable_Time_MS := 0;

    GVL_CONVERGENCE.Convergence_Lease_OK := FALSE;
    GVL_CONVERGENCE.Convergence_Release_Allowed := FALSE;

    GVL_CONVERGENCE.Convergence_Last_Healthy_MS := 0;
    GVL_CONVERGENCE.Convergence_Last_Invalidation_MS := L_Now_MS;

    GVL_CONVERGENCE.Convergence_Invalidation_Count :=
        GVL_CONVERGENCE.Convergence_Invalidation_Count + 1;

    // Oscillation quarantine.
    IF GVL_CONVERGENCE.Convergence_Invalidation_Count > 5 THEN
        GVL_CONVERGENCE.Convergence_Oscillation_Quarantine_Active := TRUE;
    END_IF;

    GVL_CONVERGENCE.Convergence_Last_Error_Code := L_Error_Code;
    GVL_CONVERGENCE.Convergence_Last_Error_Text := L_Error_Text;
END_IF;

END_PROGRAM

(* ---- PRG_CrossDomain_FailSafe_Closure_Governor.st ---- *)
PROGRAM PRG_CrossDomain_FailSafe_Closure_Governor
VAR
    L_Now_MS : UDINT;
    L_Valid : BOOL := TRUE;
END_VAR

L_Now_MS := GVL_STATUS.G_System_Time_MS;

GVL_CROSSDOMAIN_FAILSAFE_CLOSURE_FABRIC.CrossDomain_FailSafe_Closure_Valid := FALSE;
GVL_CROSSDOMAIN_FAILSAFE_CLOSURE_FABRIC.CrossDomain_FailSafe_Closure_Granted := FALSE;
GVL_CROSSDOMAIN_FAILSAFE_CLOSURE_FABRIC.CrossDomain_FailSafe_Closure_Quarantine_Active := TRUE;

IF NOT GVL_PHYSICAL_SAFESTATE_LATTICE_FABRIC.Physical_SafeState_Lattice_Granted THEN
    L_Valid := FALSE;
END_IF;

IF GVL_CROSSDOMAIN_FAILSAFE_CLOSURE_FABRIC.CrossDomain_FailSafe_Conflict_Detected
OR GVL_CROSSDOMAIN_FAILSAFE_CLOSURE_FABRIC.Unsafe_Recovery_Topology_Detected
OR GVL_CROSSDOMAIN_FAILSAFE_CLOSURE_FABRIC.CrossDomain_Recovery_Race_Detected
OR GVL_CROSSDOMAIN_FAILSAFE_CLOSURE_FABRIC.Distributed_SafeState_Fork_Detected
OR GVL_CROSSDOMAIN_FAILSAFE_CLOSURE_FABRIC.PowerDomain_Unsafe_Reactivation_Detected
OR GVL_CROSSDOMAIN_FAILSAFE_CLOSURE_FABRIC.MultiDomain_Recovery_Deadlock_Detected THEN
    L_Valid := FALSE;
END_IF;

IF L_Valid THEN
    GVL_CROSSDOMAIN_FAILSAFE_CLOSURE_FABRIC.CrossDomain_FailSafe_Closure_Valid := TRUE;
    GVL_CROSSDOMAIN_FAILSAFE_CLOSURE_FABRIC.CrossDomain_FailSafe_Closure_Granted := TRUE;
    GVL_CROSSDOMAIN_FAILSAFE_CLOSURE_FABRIC.CrossDomain_FailSafe_Closure_Quarantine_Active := FALSE;

    GVL_CROSSDOMAIN_FAILSAFE_CLOSURE_FABRIC.CrossDomain_SafeState_Compatibility_Valid := TRUE;
    GVL_CROSSDOMAIN_FAILSAFE_CLOSURE_FABRIC.FailSafe_Topology_Closure_Canonical := TRUE;
    GVL_CROSSDOMAIN_FAILSAFE_CLOSURE_FABRIC.MultiDomain_SafeTransition_Stable := TRUE;
    GVL_CROSSDOMAIN_FAILSAFE_CLOSURE_FABRIC.SafeState_Recovery_Ordering_Bounded := TRUE;
    GVL_CROSSDOMAIN_FAILSAFE_CLOSURE_FABRIC.Physical_Domain_Isolation_Coherent := TRUE;

    GVL_CROSSDOMAIN_FAILSAFE_CLOSURE_FABRIC.CrossDomain_FailSafe_Closure_Epoch :=
        GVL_PHYSICAL_SAFESTATE_LATTICE_FABRIC.Physical_SafeState_Lattice_Epoch;

    GVL_CROSSDOMAIN_FAILSAFE_CLOSURE_FABRIC.CrossDomain_FailSafe_Closure_Epoch_Coherent := TRUE;
    GVL_CROSSDOMAIN_FAILSAFE_CLOSURE_FABRIC.CrossDomain_FailSafe_Closure_Last_Update_MS := L_Now_MS;
    GVL_CROSSDOMAIN_FAILSAFE_CLOSURE_FABRIC.CrossDomain_FailSafe_Closure_Lease_Expired := FALSE;
END_IF;

END_PROGRAM

(* ---- PRG_Debug_View.st ---- *)
PROGRAM PRG_Debug_View
VAR
    L_i : INT;
    L_MaxWeight : REAL;
    L_MinWeight : REAL;
    L_Weight : REAL;
    L_Index : INT;
END_VAR

GVL_DEBUG_VIEW.D_Current_Time_MS := GVL_TIME_SERVICE.G_Now_MS;

GVL_DEBUG_VIEW.D_Safety_Mode := GVL_SAFETY_SHUTDOWN.G_Safety_Mode;
GVL_DEBUG_VIEW.D_Safety_Active := (GVL_SAFETY_SHUTDOWN.G_Safety_Mode <> NORMAL);
GVL_DEBUG_VIEW.D_Recovery_Phase := GVL_SAFETY_RECOVERY.G_Recovery_Phase;
GVL_DEBUG_VIEW.D_Recovery_Active := GVL_SAFETY_RECOVERY.G_Recovery_Active;
GVL_DEBUG_VIEW.D_Recovery_Exit_Allowed := GVL_SAFETY_RECOVERY.G_Recovery_Exit_Allowed;
GVL_DEBUG_VIEW.D_Authority_Revocation_Active := GVL_AUTHORITY_REVOCATION.Authority_Revocation_Active;
GVL_DEBUG_VIEW.D_Authority_Restoration_Allowed := GVL_AUTHORITY_RESTORATION.Authority_Restoration_Allowed;
GVL_DEBUG_VIEW.D_Authority_Restoration_Completed := GVL_AUTHORITY_RESTORATION.Authority_Restoration_Completed;

GVL_DEBUG_VIEW.D_Current_Scenario := GVL_INTENT_BEHAVIOR.I_Selected_Scenario_Text;
GVL_DEBUG_VIEW.D_Behavior_Reason := GVL_INTENT_BEHAVIOR.I_Reason_Text;

GVL_DEBUG_VIEW.D_Score_Night := GVL_INTENT_BEHAVIOR.I_Score_Night;
GVL_DEBUG_VIEW.D_Score_Preheat := GVL_INTENT_BEHAVIOR.I_Score_Preheat;
GVL_DEBUG_VIEW.D_Score_VentBoost := GVL_INTENT_BEHAVIOR.I_Score_Vent_Boost;
GVL_DEBUG_VIEW.D_Score_AccessSecure := GVL_INTENT_BEHAVIOR.I_Score_Access_Secure;

GVL_DEBUG_VIEW.D_Intent_Night := GVL_INTENT_BEHAVIOR.I_Request_Night_Mode;
GVL_DEBUG_VIEW.D_Intent_Comfort := GVL_INTENT_BEHAVIOR.I_Request_Comfort_Mode;
GVL_DEBUG_VIEW.D_Intent_VentBoost := GVL_INTENT_BEHAVIOR.I_Request_Ventilation_Boost;
GVL_DEBUG_VIEW.D_Intent_AccessSecure := GVL_INTENT_BEHAVIOR.I_Request_Access_Secure_Mode;

GVL_DEBUG_VIEW.D_Heating_Block := GVL_COMMAND_SHADOW.G_Heating_Block;
GVL_DEBUG_VIEW.D_Vent_Stop := GVL_COMMAND_SHADOW.G_Vent_Stop;
GVL_DEBUG_VIEW.D_Water_Block := GVL_COMMAND_SHADOW.G_Water_Block;
GVL_DEBUG_VIEW.D_Access_Open_Active := GVL_COMMAND_SHADOW.G_Gate_Open OR GVL_COMMAND_SHADOW.G_Wicket_Open;

GVL_DEBUG_VIEW.D_Global_Reason := GVL_EXPLAINABILITY.G_Last_Global_Reason_Text;
GVL_DEBUG_VIEW.D_Behavior_Why_Active := GVL_EXPLAINABILITY.G_Behavior_Why_Active;
GVL_DEBUG_VIEW.D_Heating_Why_Blocked := GVL_EXPLAINABILITY.G_Heating_Why_Blocked;
GVL_DEBUG_VIEW.D_Vent_Why_Stopped := GVL_EXPLAINABILITY.G_Vent_Why_Stopped;
GVL_DEBUG_VIEW.D_Water_Why_Closed := GVL_EXPLAINABILITY.G_Water_Why_Closed;
GVL_DEBUG_VIEW.D_Access_Why_Opened := GVL_EXPLAINABILITY.G_Access_Why_Opened;

// MAIN PHASE FEEDBACK SUMMARY -> DEBUG VIEW
GVL_DEBUG_VIEW.D_Main_Phase_Current := GVL_MAIN_PHASE_FEEDBACK.G_Current_Phase;
GVL_DEBUG_VIEW.D_Main_Phase_Critical_Executed := GVL_MAIN_PHASE_FEEDBACK.G_Critical_Path_Executed;
GVL_DEBUG_VIEW.D_Main_Phase_Critical_Valid := GVL_MAIN_PHASE_FEEDBACK.G_Critical_Path_Valid;
GVL_DEBUG_VIEW.D_Main_Phase_Observability_Executed := GVL_MAIN_PHASE_FEEDBACK.G_Observability_Path_Executed;
GVL_DEBUG_VIEW.D_Main_Phase_Observability_Valid := GVL_MAIN_PHASE_FEEDBACK.G_Observability_Path_Valid;
GVL_DEBUG_VIEW.D_Main_Phase_Any_Invalid := GVL_MAIN_PHASE_FEEDBACK.G_Any_Phase_Invalid;
GVL_DEBUG_VIEW.D_Main_Phase_Any_Skipped_By_Design := GVL_MAIN_PHASE_FEEDBACK.G_Any_Phase_Skipped_By_Design;
GVL_DEBUG_VIEW.D_Main_Phase_Status_Code := GVL_MAIN_PHASE_FEEDBACK.G_Status_Code;
GVL_DEBUG_VIEW.D_Main_Phase_Status_Text := GVL_MAIN_PHASE_FEEDBACK.G_Status_Text;

// DOMAIN EXECUTION POLICY SUMMARY -> DEBUG VIEW
GVL_DEBUG_VIEW.D_Domain_Policy_Any_Critical := GVL_DOMAIN_EXECUTION_POLICY.Any_Critical_Run;
GVL_DEBUG_VIEW.D_Domain_Policy_Any_Periodic := GVL_DOMAIN_EXECUTION_POLICY.Any_Periodic_Run;
GVL_DEBUG_VIEW.D_Domain_Policy_Any_Periodic_Due := GVL_DOMAIN_EXECUTION_POLICY.Any_Periodic_Due;
GVL_DEBUG_VIEW.D_Domain_Policy_Any_Idle := GVL_DOMAIN_EXECUTION_POLICY.Any_Idle_By_Design;
GVL_DEBUG_VIEW.D_Domain_Policy_Status_Code := GVL_DOMAIN_EXECUTION_POLICY.Status_Code;
GVL_DEBUG_VIEW.D_Domain_Policy_Status_Text := GVL_DOMAIN_EXECUTION_POLICY.Status_Text;

GVL_DEBUG_VIEW.D_Access_Mode := GVL_DOMAIN_EXECUTION_POLICY.Access_Mode;
GVL_DEBUG_VIEW.D_Access_Critical_Run := GVL_DOMAIN_EXECUTION_POLICY.Access_Critical_Run;
GVL_DEBUG_VIEW.D_Access_Periodic_Run := GVL_DOMAIN_EXECUTION_POLICY.Access_Periodic_Run;
GVL_DEBUG_VIEW.D_Access_Periodic_Due := GVL_DOMAIN_EXECUTION_POLICY.Access_Periodic_Due;
GVL_DEBUG_VIEW.D_Access_Idle_By_Design := GVL_DOMAIN_EXECUTION_POLICY.Access_Idle_By_Design;

GVL_DEBUG_VIEW.D_Lighting_Mode := GVL_DOMAIN_EXECUTION_POLICY.Lighting_Mode;
GVL_DEBUG_VIEW.D_Lighting_Critical_Run := GVL_DOMAIN_EXECUTION_POLICY.Lighting_Critical_Run;
GVL_DEBUG_VIEW.D_Lighting_Periodic_Run := GVL_DOMAIN_EXECUTION_POLICY.Lighting_Periodic_Run;
GVL_DEBUG_VIEW.D_Lighting_Periodic_Due := GVL_DOMAIN_EXECUTION_POLICY.Lighting_Periodic_Due;
GVL_DEBUG_VIEW.D_Lighting_Idle_By_Design := GVL_DOMAIN_EXECUTION_POLICY.Lighting_Idle_By_Design;

GVL_DEBUG_VIEW.D_Water_Mode := GVL_DOMAIN_EXECUTION_POLICY.Water_Mode;
GVL_DEBUG_VIEW.D_Water_Critical_Run := GVL_DOMAIN_EXECUTION_POLICY.Water_Critical_Run;
GVL_DEBUG_VIEW.D_Water_Periodic_Run := GVL_DOMAIN_EXECUTION_POLICY.Water_Periodic_Run;
GVL_DEBUG_VIEW.D_Water_Periodic_Due := GVL_DOMAIN_EXECUTION_POLICY.Water_Periodic_Due;
GVL_DEBUG_VIEW.D_Water_Idle_By_Design := GVL_DOMAIN_EXECUTION_POLICY.Water_Idle_By_Design;

GVL_DEBUG_VIEW.D_Heating_Mode := GVL_DOMAIN_EXECUTION_POLICY.Heating_Mode;
GVL_DEBUG_VIEW.D_Heating_Critical_Run := GVL_DOMAIN_EXECUTION_POLICY.Heating_Critical_Run;
GVL_DEBUG_VIEW.D_Heating_Periodic_Run := GVL_DOMAIN_EXECUTION_POLICY.Heating_Periodic_Run;
GVL_DEBUG_VIEW.D_Heating_Periodic_Due := GVL_DOMAIN_EXECUTION_POLICY.Heating_Periodic_Due;
GVL_DEBUG_VIEW.D_Heating_Idle_By_Design := GVL_DOMAIN_EXECUTION_POLICY.Heating_Idle_By_Design;

GVL_DEBUG_VIEW.D_Vent_Mode := GVL_DOMAIN_EXECUTION_POLICY.Vent_Mode;
GVL_DEBUG_VIEW.D_Vent_Critical_Run := GVL_DOMAIN_EXECUTION_POLICY.Vent_Critical_Run;
GVL_DEBUG_VIEW.D_Vent_Periodic_Run := GVL_DOMAIN_EXECUTION_POLICY.Vent_Periodic_Run;
GVL_DEBUG_VIEW.D_Vent_Periodic_Due := GVL_DOMAIN_EXECUTION_POLICY.Vent_Periodic_Due;
GVL_DEBUG_VIEW.D_Vent_Idle_By_Design := GVL_DOMAIN_EXECUTION_POLICY.Vent_Idle_By_Design;

GVL_DEBUG_VIEW.D_Simulation_Mode := GVL_DOMAIN_EXECUTION_POLICY.Simulation_Mode;
GVL_DEBUG_VIEW.D_Simulation_Run_Allowed := GVL_DOMAIN_EXECUTION_POLICY.Simulation_Run_Allowed;
GVL_DEBUG_VIEW.D_Simulation_Periodic_Due := GVL_DOMAIN_EXECUTION_POLICY.Simulation_Periodic_Due;
GVL_DEBUG_VIEW.D_Simulation_Idle_By_Design := GVL_DOMAIN_EXECUTION_POLICY.Simulation_Idle_By_Design;

// DOMAIN EXECUTION VALIDATION SUMMARY -> DEBUG VIEW
GVL_DEBUG_VIEW.D_Domain_Validation_Executed := GVL_DOMAIN_EXECUTION_VALIDATION.G_Validation_Executed;
GVL_DEBUG_VIEW.D_Domain_Validation_Valid := GVL_DOMAIN_EXECUTION_VALIDATION.G_Validation_Valid;
GVL_DEBUG_VIEW.D_Domain_Validation_Any_Stale_Output_Risk := GVL_DOMAIN_EXECUTION_VALIDATION.Any_Stale_Output_Risk;
GVL_DEBUG_VIEW.D_Domain_Validation_Any_Policy_Mismatch := GVL_DOMAIN_EXECUTION_VALIDATION.Any_Policy_Mismatch;
GVL_DEBUG_VIEW.D_Access_Stale_Output_Risk := GVL_DOMAIN_EXECUTION_VALIDATION.Access_Stale_Output_Risk;
GVL_DEBUG_VIEW.D_Lighting_Stale_Output_Risk := GVL_DOMAIN_EXECUTION_VALIDATION.Lighting_Stale_Output_Risk;
GVL_DEBUG_VIEW.D_Water_Stale_Output_Risk := GVL_DOMAIN_EXECUTION_VALIDATION.Water_Stale_Output_Risk;
GVL_DEBUG_VIEW.D_Heating_Stale_Output_Risk := GVL_DOMAIN_EXECUTION_VALIDATION.Heating_Stale_Output_Risk;
GVL_DEBUG_VIEW.D_Vent_Stale_Output_Risk := GVL_DOMAIN_EXECUTION_VALIDATION.Vent_Stale_Output_Risk;
GVL_DEBUG_VIEW.D_Domain_Validation_Status_Code := GVL_DOMAIN_EXECUTION_VALIDATION.Status_Code;
GVL_DEBUG_VIEW.D_Domain_Validation_Status_Text := GVL_DOMAIN_EXECUTION_VALIDATION.Status_Text;

// RUNTIME SCENARIO VALIDATION SUMMARY -> DEBUG VIEW
GVL_DEBUG_VIEW.D_Runtime_Scenario_Validation_Executed := GVL_RUNTIME_SCENARIO_VALIDATION.G_Validation_Executed;
GVL_DEBUG_VIEW.D_Runtime_Scenario_Validation_Valid := GVL_RUNTIME_SCENARIO_VALIDATION.G_Validation_Valid;
GVL_DEBUG_VIEW.D_Runtime_Scenario_Any_Context_Invalid := GVL_RUNTIME_SCENARIO_VALIDATION.Any_Context_Invalid;
GVL_DEBUG_VIEW.D_Runtime_Idle_Context_Active := GVL_RUNTIME_SCENARIO_VALIDATION.Idle_Context_Active;
GVL_DEBUG_VIEW.D_Runtime_Security_Context_Active := GVL_RUNTIME_SCENARIO_VALIDATION.Security_Context_Active;
GVL_DEBUG_VIEW.D_Runtime_Away_Context_Active := GVL_RUNTIME_SCENARIO_VALIDATION.Away_Context_Active;
GVL_DEBUG_VIEW.D_Runtime_Presence_Context_Active := GVL_RUNTIME_SCENARIO_VALIDATION.Presence_Context_Active;
GVL_DEBUG_VIEW.D_Runtime_Fire_Context_Active := GVL_RUNTIME_SCENARIO_VALIDATION.Fire_Context_Active;
GVL_DEBUG_VIEW.D_Runtime_Gas_Context_Active := GVL_RUNTIME_SCENARIO_VALIDATION.Gas_Context_Active;
GVL_DEBUG_VIEW.D_Runtime_Leak_Context_Active := GVL_RUNTIME_SCENARIO_VALIDATION.Leak_Context_Active;
GVL_DEBUG_VIEW.D_Runtime_Global_Stop_Context_Active := GVL_RUNTIME_SCENARIO_VALIDATION.Global_Stop_Context_Active;
GVL_DEBUG_VIEW.D_Runtime_Freeze_Context_Active := GVL_RUNTIME_SCENARIO_VALIDATION.Freeze_Context_Active;
GVL_DEBUG_VIEW.D_Runtime_Heating_Context_Valid := GVL_RUNTIME_SCENARIO_VALIDATION.Heating_Context_Valid;
GVL_DEBUG_VIEW.D_Runtime_Vent_Context_Valid := GVL_RUNTIME_SCENARIO_VALIDATION.Vent_Context_Valid;
GVL_DEBUG_VIEW.D_Runtime_Access_Context_Valid := GVL_RUNTIME_SCENARIO_VALIDATION.Access_Context_Valid;
GVL_DEBUG_VIEW.D_Runtime_Global_Stop_Context_Valid := GVL_RUNTIME_SCENARIO_VALIDATION.Global_Stop_Context_Valid;
GVL_DEBUG_VIEW.D_Runtime_Scenario_Status_Code := GVL_RUNTIME_SCENARIO_VALIDATION.Status_Code;
GVL_DEBUG_VIEW.D_Runtime_Scenario_Status_Text := GVL_RUNTIME_SCENARIO_VALIDATION.Status_Text;

// RUNTIME PHYSICAL IO VALIDATION SUMMARY -> DEBUG VIEW
GVL_DEBUG_VIEW.D_Runtime_IO_Validation_Executed := GVL_RUNTIME_IO_VALIDATION.G_Validation_Executed;
GVL_DEBUG_VIEW.D_Runtime_IO_Validation_Valid := GVL_RUNTIME_IO_VALIDATION.G_Validation_Valid;
GVL_DEBUG_VIEW.D_Runtime_IO_Any_Invalid := GVL_RUNTIME_IO_VALIDATION.Any_IO_Invalid;
GVL_DEBUG_VIEW.D_Runtime_IO_Fire_Valid := GVL_RUNTIME_IO_VALIDATION.Fire_IO_Valid;
GVL_DEBUG_VIEW.D_Runtime_IO_Gas_Valid := GVL_RUNTIME_IO_VALIDATION.Gas_IO_Valid;
GVL_DEBUG_VIEW.D_Runtime_IO_Leak_Valid := GVL_RUNTIME_IO_VALIDATION.Leak_IO_Valid;
GVL_DEBUG_VIEW.D_Runtime_IO_Global_Stop_Valid := GVL_RUNTIME_IO_VALIDATION.Global_Stop_IO_Valid;
GVL_DEBUG_VIEW.D_Runtime_IO_Inactive_PLC_Valid := GVL_RUNTIME_IO_VALIDATION.Inactive_PLC_IO_Valid;
GVL_DEBUG_VIEW.D_Runtime_IO_Freeze_Valid := GVL_RUNTIME_IO_VALIDATION.Freeze_IO_Valid;
GVL_DEBUG_VIEW.D_Runtime_IO_Status_Code := GVL_RUNTIME_IO_VALIDATION.Status_Code;
GVL_DEBUG_VIEW.D_Runtime_IO_Status_Text := GVL_RUNTIME_IO_VALIDATION.Status_Text;

// SENSOR QUALITY → HMI
GVL_DEBUG_VIEW.D_Input_Source_Valid := GVL_INPUT.IN_Source_Valid;
GVL_DEBUG_VIEW.D_Input_Degraded := GVL_INPUT.IN_Input_Degraded;
GVL_DEBUG_VIEW.D_Sensor_Fault := GVL_INPUT.IN_Sensor_Fault;
GVL_DEBUG_VIEW.D_Validation_Failed := GVL_INPUT.IN_Validation_Failed;
GVL_DEBUG_VIEW.D_Anomaly_Detected := GVL_INPUT.IN_Anomaly_Detected;
GVL_DEBUG_VIEW.D_Validation_Reason := GVL_INPUT.IN_Validation_Reason;
GVL_DEBUG_VIEW.D_Anomaly_Reason := GVL_INPUT.IN_Anomaly_Reason;
GVL_DEBUG_VIEW.D_Last_Invalid_Zone := GVL_INPUT.IN_Last_Invalid_Zone;
GVL_DEBUG_VIEW.D_Min_Zone_Confidence := GVL_INPUT.IN_Min_Zone_Confidence;
GVL_DEBUG_VIEW.D_Worst_Zone := GVL_INPUT.IN_Worst_Zone;

GVL_DEBUG_VIEW.D_Adapt_Profile := GVL_BEHAVIOR_ADAPT.G_Adapt_Profile;

IF GVL_BEHAVIOR_ADAPT.G_Adapt_Profile = ADAPT_PROFILE_STABLE THEN
    GVL_DEBUG_VIEW.D_Adapt_Profile_Text := 'STABLE';
ELSIF GVL_BEHAVIOR_ADAPT.G_Adapt_Profile = ADAPT_PROFILE_BALANCED THEN
    GVL_DEBUG_VIEW.D_Adapt_Profile_Text := 'BALANCED';
ELSE
    GVL_DEBUG_VIEW.D_Adapt_Profile_Text := 'AGGRESSIVE';
END_IF;

L_MaxWeight := 0.0;
L_MinWeight := 9999.0;
GVL_DEBUG_VIEW.D_Main_VentBoost_Zone := 0;

FOR L_i := 1 TO GVL_CONSTANTS.C_MAX_ZONES DO
    L_Weight := GVL_BEHAVIOR_ADAPT.G_VentBoost_Zone_Adapt[L_i].Zone_Weight;
    IF L_Weight > L_MaxWeight THEN
        L_MaxWeight := L_Weight;
        GVL_DEBUG_VIEW.D_Main_VentBoost_Zone := L_i;
        GVL_DEBUG_VIEW.D_Main_VentBoost_Zone_Weight := L_Weight;
        GVL_DEBUG_VIEW.D_Main_VentBoost_Zone_Confidence :=
            GVL_BEHAVIOR_ADAPT.G_VentBoost_Zone_Adapt[L_i].Confidence;
    END_IF;
    IF L_Weight < L_MinWeight THEN
        L_MinWeight := L_Weight;
    END_IF;
END_FOR;

GVL_DEBUG_VIEW.D_Max_VentBoost_Zone_Weight := L_MaxWeight;
GVL_DEBUG_VIEW.D_Min_VentBoost_Zone_Weight := L_MinWeight;

L_Index := GVL_TRACE.G_Trace_Write_Index - 1;
IF L_Index < 1 THEN
    L_Index := 200;
END_IF;

GVL_DEBUG_VIEW.D_Last_Trace_Text := GVL_TRACE.G_Trace_Buffer[L_Index].Text;
GVL_DEBUG_VIEW.D_Last_Trace_Time_MS := GVL_TRACE.G_Trace_Buffer[L_Index].Timestamp_MS;
GVL_DEBUG_VIEW.D_Last_Trace_Reason := GVL_TRACE.G_Trace_Buffer[L_Index].Reason_Code;

END_PROGRAM

(* ---- PRG_Distributed_Commit_Governor.st ---- *)
PROGRAM PRG_Distributed_Commit_Governor
VAR
    L_Now_MS : UDINT;
    L_Delta_MS : UDINT;
    L_Commit_Valid : BOOL := TRUE;
    L_Error_Code : UDINT := 0;
    L_Error_Text : STRING(160) := '';
    L_Peer_Session_Active : BOOL := FALSE;

    L_Publication_Authority_Allowed : BOOL;
END_VAR

L_Now_MS := GVL_STATUS.G_System_Time_MS;
L_Commit_Valid := TRUE;
L_Error_Code := 0;
L_Error_Text := '';

GVL_DISTRIBUTED_COMMIT.Peer_Commit_Ack_Expired := FALSE;
GVL_DISTRIBUTED_COMMIT.Peer_Commit_Mismatch := FALSE;
GVL_DISTRIBUTED_COMMIT.Peer_Commit_Replay_Detected := FALSE;
GVL_DISTRIBUTED_COMMIT.Peer_Commit_Missing := FALSE;
GVL_DISTRIBUTED_COMMIT.Commit_Lease_Expired := FALSE;

L_Publication_Authority_Allowed :=
    GVL_Distributed_Execution_Gates.G_Runtime_Valid
    AND GVL_Distributed_Execution_Gates.G_Can_Replicate
    AND GVL_Distributed_Execution_Gates.G_Can_Own_Projection
    AND GVL_CONVERGENCE.Convergence_Lease_OK
    AND GVL_CONVERGENCE.Convergence_Release_Allowed
    AND GVL_RECOVERY_GOVERNANCE.Recovery_Governance_Valid
    AND NOT GVL_RECOVERY_GOVERNANCE.Recovery_Quarantine_Active;

GVL_DISTRIBUTED_COMMIT.Local_Publication_Commit_Epoch := GVL_DISTRIBUTED_SNAPSHOT.Distributed_Snapshot_Epoch;
GVL_DISTRIBUTED_COMMIT.Local_Prepare_Epoch := GVL_DISTRIBUTED_SNAPSHOT.Distributed_Snapshot_Epoch;

IF NOT L_Publication_Authority_Allowed THEN
    L_Commit_Valid := FALSE;
    L_Error_Code := 14999;
    L_Error_Text := 'Distributed publication authority restricted';
END_IF;

IF L_Commit_Valid THEN
    IF GVL_DISTRIBUTED_SNAPSHOT.Distributed_Publication_Reconciled
    AND GVL_DISTRIBUTED_SNAPSHOT.Distributed_Publication_Freeze_Valid
    AND GVL_DISTRIBUTED_SNAPSHOT.Distributed_Snapshot_Consistent
    THEN
        GVL_DISTRIBUTED_COMMIT.Publication_Prepare_Active := TRUE;
        GVL_DISTRIBUTED_COMMIT.Publication_Prepare_Valid := TRUE;
    ELSE
        GVL_DISTRIBUTED_COMMIT.Publication_Prepare_Active := FALSE;
        GVL_DISTRIBUTED_COMMIT.Publication_Prepare_Valid := FALSE;
        L_Commit_Valid := FALSE;
        L_Error_Code := 15000;
        L_Error_Text := 'Distributed immutable publication prepare invalid';
    END_IF;
END_IF;

IF GVL_DISTRIBUTED_COMMIT.Peer_Publication_Commit_Epoch > 0 THEN
    L_Peer_Session_Active := TRUE;
END_IF;

IF GVL_DISTRIBUTED_COMMIT.Peer_Prepare_Epoch > 0 THEN
    L_Peer_Session_Active := TRUE;
END_IF;

IF GVL_DISTRIBUTED_COMMIT.Peer_Commit_Ack_Valid THEN
    L_Peer_Session_Active := TRUE;
END_IF;

IF L_Commit_Valid AND L_Peer_Session_Active THEN
    L_Delta_MS := L_Now_MS - GVL_DISTRIBUTED_COMMIT.Peer_Commit_Last_Refresh_MS;

    IF GVL_DISTRIBUTED_COMMIT.Commit_Lease_Active THEN
        IF L_Delta_MS > GVL_DISTRIBUTED_COMMIT.Commit_Timeout_MS THEN
            GVL_DISTRIBUTED_COMMIT.Commit_Lease_Expired := TRUE;
            L_Commit_Valid := FALSE;
            L_Error_Code := 15001;
            L_Error_Text := 'Distributed commit lease expired';
        END_IF;
    END_IF;
END_IF;

IF L_Commit_Valid AND L_Peer_Session_Active THEN
    IF NOT GVL_DISTRIBUTED_COMMIT.Peer_Commit_Ack_Valid THEN
        GVL_DISTRIBUTED_COMMIT.Peer_Commit_Missing := TRUE;
        L_Commit_Valid := FALSE;
        L_Error_Code := 15002;
        L_Error_Text := 'Peer commit acknowledgement missing';
    END_IF;
END_IF;

IF L_Commit_Valid AND L_Peer_Session_Active THEN
    IF GVL_DISTRIBUTED_COMMIT.Peer_Publication_Commit_Epoch < GVL_DISTRIBUTED_COMMIT.Local_Publication_Commit_Epoch THEN
        GVL_DISTRIBUTED_COMMIT.Peer_Commit_Mismatch := TRUE;
        L_Commit_Valid := FALSE;
        L_Error_Code := 15003;
        L_Error_Text := 'Peer commit epoch mismatch';
    END_IF;
END_IF;

IF L_Commit_Valid AND L_Peer_Session_Active THEN
    IF GVL_DISTRIBUTED_COMMIT.Peer_Prepare_Epoch < GVL_DISTRIBUTED_COMMIT.Local_Prepare_Epoch THEN
        GVL_DISTRIBUTED_COMMIT.Peer_Commit_Replay_Detected := TRUE;
        L_Commit_Valid := FALSE;
        L_Error_Code := 15004;
        L_Error_Text := 'Peer commit replay detected';
    END_IF;
END_IF;

IF L_Commit_Valid THEN
    GVL_DISTRIBUTED_COMMIT.Distributed_Commit_Epoch := GVL_DISTRIBUTED_COMMIT.Distributed_Commit_Epoch + 1;
    GVL_DISTRIBUTED_COMMIT.Distributed_Commit_Reconciliation_Epoch := GVL_DISTRIBUTED_COMMIT.Distributed_Commit_Reconciliation_Epoch + 1;

    GVL_DISTRIBUTED_COMMIT.Publication_Commit_Requested := TRUE;
    GVL_DISTRIBUTED_COMMIT.Publication_Commit_Confirmed := TRUE;

    IF L_Peer_Session_Active THEN
        GVL_DISTRIBUTED_COMMIT.Commit_Lease_Active := TRUE;
    ELSE
        GVL_DISTRIBUTED_COMMIT.Commit_Lease_Active := FALSE;
    END_IF;

    GVL_DISTRIBUTED_COMMIT.Distributed_Commit_Valid := TRUE;

    IF GVL_CONVERGENCE.Convergence_Release_Allowed THEN
        GVL_DISTRIBUTED_COMMIT.Distributed_Commit_Quarantine_Active := FALSE;
    END_IF;

    GVL_DISTRIBUTED_COMMIT.Commit_Last_Reconciliation_MS := L_Now_MS;
    GVL_DISTRIBUTED_COMMIT.Distributed_Commit_Last_Error_Code := 0;
    GVL_DISTRIBUTED_COMMIT.Distributed_Commit_Last_Error_Text := '';
ELSE
    GVL_DISTRIBUTED_COMMIT.Publication_Commit_Confirmed := FALSE;
    GVL_DISTRIBUTED_COMMIT.Distributed_Commit_Valid := FALSE;
    GVL_DISTRIBUTED_COMMIT.Distributed_Commit_Quarantine_Active := TRUE;
    GVL_DISTRIBUTED_COMMIT.Distributed_Commit_Last_Error_Code := L_Error_Code;
    GVL_DISTRIBUTED_COMMIT.Distributed_Commit_Last_Error_Text := L_Error_Text;
END_IF;
END_PROGRAM

(* ---- PRG_Distributed_Domain.st ---- *)
PROGRAM PRG_Distributed_Domain
// CANONICAL EXECUTION DOMAIN
// PRESERVES EXECUTION ORDER

PRG_Distributed_Peer_Ingestion();
PRG_Distributed_Epoch_Governor();
PRG_Distributed_Snapshot_Governor();
PRG_Distributed_Runtime_Supervisor();
PRG_Distributed_Commit_Governor();

END_PROGRAM

(* ---- PRG_Distributed_Epoch_Linearity_Governor.st ---- *)
PROGRAM PRG_Distributed_Epoch_Linearity_Governor
IF GVL_TEMPORAL_CAUSALITY_CLOSURE_FABRIC.Temporal_Causality_Closure_Granted
AND NOT GVL_DISTRIBUTED_EPOCH_LINEARITY_FABRIC.Epoch_Rollback_Detected
AND NOT GVL_DISTRIBUTED_EPOCH_LINEARITY_FABRIC.Distributed_Epoch_Fork_Detected
AND NOT GVL_DISTRIBUTED_EPOCH_LINEARITY_FABRIC.Stale_Epoch_Application_Detected THEN

    GVL_DISTRIBUTED_EPOCH_LINEARITY_FABRIC.Distributed_Epoch_Linearity_Valid := TRUE;
    GVL_DISTRIBUTED_EPOCH_LINEARITY_FABRIC.Distributed_Epoch_Linearity_Granted := TRUE;
    GVL_DISTRIBUTED_EPOCH_LINEARITY_FABRIC.Distributed_Epoch_Linearity_Valid_Proof := TRUE;
    GVL_DISTRIBUTED_EPOCH_LINEARITY_FABRIC.Epoch_Timeline_Monotonic := TRUE;
    GVL_DISTRIBUTED_EPOCH_LINEARITY_FABRIC.Cluster_Epoch_Consensus_Stable := TRUE;
END_IF;
END_PROGRAM

(* ---- PRG_Distributed_Forward_Progress_Governor.st ---- *)
PROGRAM PRG_Distributed_Forward_Progress_Governor
IF GVL_RESOURCE_STARVATION_BOUNDARY_FABRIC.Resource_Starvation_Boundary_Granted
AND NOT GVL_DISTRIBUTED_FORWARD_PROGRESS_FABRIC.Distributed_Livelock_Detected
AND NOT GVL_DISTRIBUTED_FORWARD_PROGRESS_FABRIC.Cluster_Progress_Fork_Detected
AND NOT GVL_DISTRIBUTED_FORWARD_PROGRESS_FABRIC.Distributed_Consensus_Progress_Deadlock THEN

    GVL_DISTRIBUTED_FORWARD_PROGRESS_FABRIC.Distributed_Forward_Progress_Valid := TRUE;
    GVL_DISTRIBUTED_FORWARD_PROGRESS_FABRIC.Distributed_Forward_Progress_Granted := TRUE;
    GVL_DISTRIBUTED_FORWARD_PROGRESS_FABRIC.Distributed_Forward_Progress_Canonical := TRUE;
    GVL_DISTRIBUTED_FORWARD_PROGRESS_FABRIC.Cluster_Progress_Consensus_Stable := TRUE;
    GVL_DISTRIBUTED_FORWARD_PROGRESS_FABRIC.Distributed_Recovery_Progress_Valid := TRUE;
END_IF;
END_PROGRAM

(* ---- PRG_Distributed_Peer_Ingestion.st ---- *)
PROGRAM PRG_Distributed_Peer_Ingestion
VAR
    L_Now_MS : UDINT;
END_VAR

// ======================================================
// DISTRIBUTED PEER INGESTION
// ======================================================
// Bounded peer-session ingestion layer.
//
// Purpose:
// normalize replicated HA session state into distributed
// peer-input fields consumed by distributed governors.
//
// This layer does NOT:
// - perform reconciliation/quarantine decisions
// - perform split-brain detection
// - validate peer publication correctness
// - mutate local runtime authority
// ======================================================

L_Now_MS := GVL_STATUS.G_System_Time_MS;

// ------------------------------------------------------
// Peer session freshness projection.
// ------------------------------------------------------

GVL_DISTRIBUTED_EPOCH.Peer_Last_Refresh_MS :=
    GVL_HA_SESSION_REPLICATION.HA_Remote_Last_Refresh_MS;

GVL_DISTRIBUTED_EPOCH.Peer_Lease_Active :=
    GVL_HA_SESSION_REPLICATION.HA_Remote_Session_Valid;

// ------------------------------------------------------
// Replicated remote session ingestion.
// ------------------------------------------------------

IF GVL_HA_SESSION_REPLICATION.HA_Remote_Session_Valid THEN
    GVL_DISTRIBUTED_EPOCH.Peer_Runtime_Epoch :=
        GVL_HA_SESSION_REPLICATION.HA_Remote_Runtime_Epoch;

    GVL_DISTRIBUTED_EPOCH.Peer_Snapshot_Epoch :=
        GVL_HA_SESSION_REPLICATION.HA_Remote_Snapshot_Epoch;

    GVL_DISTRIBUTED_EPOCH.Peer_Boot_Generation :=
        GVL_HA_SESSION_REPLICATION.HA_Remote_Boot_Generation;

    GVL_DISTRIBUTED_EPOCH.Peer_Fencing_Token :=
        GVL_HA_SESSION_REPLICATION.HA_Remote_Fencing_Token;
ELSE
    GVL_DISTRIBUTED_EPOCH.Peer_Lease_Active := FALSE;
    GVL_DISTRIBUTED_EPOCH.Peer_Runtime_Epoch := 0;
    GVL_DISTRIBUTED_EPOCH.Peer_Snapshot_Epoch := 0;
    GVL_DISTRIBUTED_EPOCH.Peer_Boot_Generation := 0;
    GVL_DISTRIBUTED_EPOCH.Peer_Fencing_Token := 0;
    GVL_DISTRIBUTED_EPOCH.Peer_Last_Refresh_MS := 0;
END_IF;

// >>> BULK_SYNC_ANCHOR: PRG_Distributed_Peer_Ingestion <<<
END_PROGRAM

(* ---- PRG_Distributed_Snapshot_Governor.st ---- *)
PROGRAM PRG_Distributed_Snapshot_Governor
VAR
    L_Now_MS : UDINT;
    L_Delta_MS : UDINT;
    L_Distributed_Snapshot_Valid : BOOL := TRUE;
    L_Error_Code : UDINT := 0;
    L_Error_Text : STRING(160) := '';
    L_Peer_Session_Active : BOOL := FALSE;
END_VAR

L_Now_MS := GVL_STATUS.G_System_Time_MS;
L_Distributed_Snapshot_Valid := TRUE;
L_Error_Code := 0;
L_Error_Text := '';

// ======================================================
// DISTRIBUTED IMMUTABLE SNAPSHOT GOVERNOR
// ======================================================
// Governs immutable peer publication snapshot exchange.
// Publication-authoritative only.
// Does not invalidate runtime barrier, PLC fencing
// or local immutable snapshot freeze.
//
// Recovery/release is convergence-lease based:
// distributed snapshot quarantine is not released on a
// single healthy scan.
// ======================================================

GVL_DISTRIBUTED_SNAPSHOT.Peer_Publication_Stale := FALSE;
GVL_DISTRIBUTED_SNAPSHOT.Peer_Snapshot_Not_Immutable := FALSE;
GVL_DISTRIBUTED_SNAPSHOT.Peer_Publication_Divergence := FALSE;
GVL_DISTRIBUTED_SNAPSHOT.Peer_Publication_Reconciliation_Lost := FALSE;
GVL_DISTRIBUTED_SNAPSHOT.Peer_Snapshot_Lease_Expired := FALSE;

// ------------------------------------------------------
// Local immutable publication projection.
// ------------------------------------------------------
// Distributed snapshot is upstream of output freshness in MAIN.
// Therefore local publication baseline must not read GVL_OUTPUT_EPOCH.
// It uses the already-frozen runtime snapshot epoch instead.
// ------------------------------------------------------

GVL_DISTRIBUTED_SNAPSHOT.Local_Distributed_Snapshot_Epoch := GVL_DISTRIBUTED_SNAPSHOT.Distributed_Snapshot_Epoch;
GVL_DISTRIBUTED_SNAPSHOT.Local_Runtime_Snapshot_Epoch := GVL_RUNTIME_SNAPSHOT.Snapshot_Epoch;
GVL_DISTRIBUTED_SNAPSHOT.Local_Publication_Epoch := GVL_RUNTIME_SNAPSHOT.Snapshot_Publication_Epoch;

// ------------------------------------------------------
// Local immutable publication freeze semantics.
// ------------------------------------------------------

IF GVL_RUNTIME_SNAPSHOT.Snapshot_Frozen
AND GVL_RUNTIME_SNAPSHOT.Snapshot_Publication_Allowed
AND GVL_RUNTIME_SNAPSHOT.Snapshot_Copy_Valid
AND GVL_RUNTIME_SNAPSHOT.Snapshot_Isolation_Valid
THEN
    GVL_DISTRIBUTED_SNAPSHOT.Distributed_Snapshot_Frozen := TRUE;
ELSE
    GVL_DISTRIBUTED_SNAPSHOT.Distributed_Snapshot_Frozen := FALSE;

    L_Distributed_Snapshot_Valid := FALSE;
    L_Error_Code := 14000;
    L_Error_Text := 'Local immutable snapshot not frozen';
END_IF;

// ------------------------------------------------------
// Peer session detection.
// ------------------------------------------------------

IF GVL_DISTRIBUTED_SNAPSHOT.Peer_Publication_Epoch > 0 THEN
    L_Peer_Session_Active := TRUE;
END_IF;

IF GVL_DISTRIBUTED_SNAPSHOT.Peer_Runtime_Snapshot_Epoch > 0 THEN
    L_Peer_Session_Active := TRUE;
END_IF;

IF GVL_DISTRIBUTED_SNAPSHOT.Peer_Distributed_Snapshot_Epoch > 0 THEN
    L_Peer_Session_Active := TRUE;
END_IF;

IF GVL_DISTRIBUTED_SNAPSHOT.Peer_Snapshot_Immutable THEN
    L_Peer_Session_Active := TRUE;
END_IF;

// ------------------------------------------------------
// Peer snapshot lease validation.
// ------------------------------------------------------

IF L_Distributed_Snapshot_Valid AND L_Peer_Session_Active THEN
    L_Delta_MS := L_Now_MS - GVL_DISTRIBUTED_SNAPSHOT.Peer_Snapshot_Last_Refresh_MS;

    IF GVL_DISTRIBUTED_SNAPSHOT.Peer_Snapshot_Lease_Active THEN
        IF L_Delta_MS > GVL_DISTRIBUTED_SNAPSHOT.Peer_Snapshot_Lease_Timeout_MS THEN
            GVL_DISTRIBUTED_SNAPSHOT.Peer_Snapshot_Lease_Expired := TRUE;

            L_Distributed_Snapshot_Valid := FALSE;
            L_Error_Code := 14001;
            L_Error_Text := 'Peer snapshot lease expired';
        END_IF;
    END_IF;
END_IF;

// ------------------------------------------------------
// Peer immutable snapshot semantics.
// ------------------------------------------------------

IF L_Distributed_Snapshot_Valid AND L_Peer_Session_Active THEN
    IF NOT GVL_DISTRIBUTED_SNAPSHOT.Peer_Snapshot_Immutable THEN
        GVL_DISTRIBUTED_SNAPSHOT.Peer_Snapshot_Not_Immutable := TRUE;

        L_Distributed_Snapshot_Valid := FALSE;
        L_Error_Code := 14002;
        L_Error_Text := 'Peer snapshot not immutable';
    END_IF;
END_IF;

// ------------------------------------------------------
// Peer publication continuity.
// ------------------------------------------------------

IF L_Distributed_Snapshot_Valid AND L_Peer_Session_Active THEN
    IF GVL_DISTRIBUTED_SNAPSHOT.Peer_Publication_Epoch < GVL_DISTRIBUTED_SNAPSHOT.Local_Publication_Epoch THEN
        GVL_DISTRIBUTED_SNAPSHOT.Peer_Publication_Stale := TRUE;
    END_IF;
END_IF;

// ------------------------------------------------------
// Peer publication reconciliation continuity.
// ------------------------------------------------------

IF L_Distributed_Snapshot_Valid AND L_Peer_Session_Active THEN
    IF GVL_DISTRIBUTED_SNAPSHOT.Peer_Runtime_Snapshot_Epoch <> GVL_DISTRIBUTED_SNAPSHOT.Local_Runtime_Snapshot_Epoch THEN
        GVL_DISTRIBUTED_SNAPSHOT.Peer_Publication_Divergence := TRUE;
    END_IF;
END_IF;

IF GVL_DISTRIBUTED_SNAPSHOT.Peer_Publication_Stale
OR GVL_DISTRIBUTED_SNAPSHOT.Peer_Publication_Divergence
OR GVL_DISTRIBUTED_SNAPSHOT.Peer_Snapshot_Not_Immutable
THEN
    GVL_DISTRIBUTED_SNAPSHOT.Peer_Publication_Reconciliation_Lost := TRUE;
END_IF;

// ------------------------------------------------------
// Publish authoritative distributed snapshot state.
// ------------------------------------------------------

IF L_Distributed_Snapshot_Valid THEN
    GVL_DISTRIBUTED_SNAPSHOT.Distributed_Snapshot_Epoch := GVL_DISTRIBUTED_SNAPSHOT.Distributed_Snapshot_Epoch + 1;
    GVL_DISTRIBUTED_SNAPSHOT.Distributed_Snapshot_Reconciliation_Epoch := GVL_DISTRIBUTED_SNAPSHOT.Distributed_Snapshot_Reconciliation_Epoch + 1;

    GVL_DISTRIBUTED_SNAPSHOT.Distributed_Publication_Reconciled := TRUE;
    GVL_DISTRIBUTED_SNAPSHOT.Distributed_Publication_Freeze_Valid := TRUE;
    GVL_DISTRIBUTED_SNAPSHOT.Distributed_Snapshot_Consistent := TRUE;

    // Lease-based recovery release.
    IF GVL_CONVERGENCE.Convergence_Release_Allowed THEN
        GVL_DISTRIBUTED_SNAPSHOT.Distributed_Snapshot_Quarantine_Active := FALSE;
    END_IF;

    GVL_DISTRIBUTED_SNAPSHOT.Distributed_Snapshot_Last_Error_Code := 0;
    GVL_DISTRIBUTED_SNAPSHOT.Distributed_Snapshot_Last_Error_Text := '';
ELSE
    // Invalid distributed snapshot state escalates immediately.
    GVL_DISTRIBUTED_SNAPSHOT.Distributed_Publication_Reconciled := FALSE;
    GVL_DISTRIBUTED_SNAPSHOT.Distributed_Publication_Freeze_Valid := FALSE;
    GVL_DISTRIBUTED_SNAPSHOT.Distributed_Snapshot_Consistent := FALSE;

    GVL_DISTRIBUTED_SNAPSHOT.Distributed_Snapshot_Quarantine_Active := TRUE;

    GVL_DISTRIBUTED_SNAPSHOT.Distributed_Snapshot_Last_Error_Code := L_Error_Code;
    GVL_DISTRIBUTED_SNAPSHOT.Distributed_Snapshot_Last_Error_Text := L_Error_Text;
END_IF;
END_PROGRAM

(* ---- PRG_Distributed_Snapshot_Ingestion.st ---- *)
PROGRAM PRG_Distributed_Snapshot_Ingestion
// ======================================================
// DISTRIBUTED SNAPSHOT INGESTION
// ======================================================
// Canonical replicated distributed snapshot ingestion.
//
// Purpose:
// normalize replicated immutable snapshot state from
// HA/session replication boundary into peer snapshot fields.
//
// This layer does NOT:
// - perform distributed reconciliation
// - mutate local runtime snapshot authority
// - mutate output/runtime authority
// ======================================================

IF NOT GVL_HA_SESSION_REPLICATION.HA_Remote_Session_Valid THEN
    GVL_DISTRIBUTED_SNAPSHOT.Peer_Distributed_Snapshot_Epoch := 0;
    GVL_DISTRIBUTED_SNAPSHOT.Peer_Runtime_Snapshot_Epoch := 0;
    GVL_DISTRIBUTED_SNAPSHOT.Peer_Publication_Epoch := 0;

    GVL_DISTRIBUTED_SNAPSHOT.Peer_Snapshot_Immutable := FALSE;
    GVL_DISTRIBUTED_SNAPSHOT.Peer_Snapshot_Lease_Active := FALSE;
    GVL_DISTRIBUTED_SNAPSHOT.Peer_Snapshot_Last_Refresh_MS := 0;

    RETURN;
END_IF;

GVL_DISTRIBUTED_SNAPSHOT.Peer_Distributed_Snapshot_Epoch :=
    GVL_HA_SESSION_REPLICATION.HA_Remote_Distributed_Snapshot_Epoch;

GVL_DISTRIBUTED_SNAPSHOT.Peer_Runtime_Snapshot_Epoch :=
    GVL_HA_SESSION_REPLICATION.HA_Remote_Runtime_Snapshot_Epoch;

GVL_DISTRIBUTED_SNAPSHOT.Peer_Publication_Epoch :=
    GVL_HA_SESSION_REPLICATION.HA_Remote_Publication_Epoch;

GVL_DISTRIBUTED_SNAPSHOT.Peer_Snapshot_Immutable :=
    GVL_HA_SESSION_REPLICATION.HA_Remote_Snapshot_Immutable;

GVL_DISTRIBUTED_SNAPSHOT.Peer_Snapshot_Lease_Active := TRUE;

GVL_DISTRIBUTED_SNAPSHOT.Peer_Snapshot_Last_Refresh_MS :=
    GVL_HA_SESSION_REPLICATION.HA_Remote_Snapshot_Last_Refresh_MS;

// >>> BULK_SYNC_ANCHOR: PRG_Distributed_Snapshot_Ingestion <<<
END_PROGRAM

(* ---- PRG_Domain_Execution_Policy.st ---- *)
PROGRAM PRG_Domain_Execution_Policy
// Observational domain execution policy.
// Classifies domains as critical, periodic or idle-by-design.
// Does not gate execution and does not write physical outputs.
VAR
    L_i : INT;
    L_Heating_Output_Active : BOOL;
    L_Vent_Output_Active : BOOL;
END_VAR

GVL_DOMAIN_EXECUTION_POLICY.G_Last_Update_MS := GVL_TIME_SERVICE.G_Now_MS;

GVL_DOMAIN_EXECUTION_POLICY.G_Security_Context_Active :=
    GVL_ALARM.G_Security_Armed
    OR GVL_ALARM.G_Security_Alarm;

GVL_DOMAIN_EXECUTION_POLICY.G_Away_Context_Active :=
    GVL_STATUS.G_Current_Scenario = SCENARIO_AWAY;

GVL_DOMAIN_EXECUTION_POLICY.G_Presence_Context_Active :=
    GVL_STATUS.G_Current_Scenario = SCENARIO_PRESENCE;

GVL_DOMAIN_EXECUTION_POLICY.G_Emergency_Context_Active :=
    (GVL_SAFETY_SHUTDOWN.G_Safety_Mode = FIRE)
    OR (GVL_SAFETY_SHUTDOWN.G_Safety_Mode = GAS)
    OR (GVL_SAFETY_SHUTDOWN.G_Safety_Mode = WATER_LEAK)
    OR (GVL_SAFETY_SHUTDOWN.G_Safety_Mode = GLOBAL_STOP);

GVL_DOMAIN_EXECUTION_POLICY.Access_Critical_Run :=
    (GVL_SAFETY_SHUTDOWN.G_Safety_Mode = FIRE)
    OR (GVL_SAFETY_SHUTDOWN.G_Safety_Mode = GAS)
    OR GVL_COMMAND_SHADOW.G_Lock_1_Open
    OR GVL_COMMAND_SHADOW.G_Lock_1_Close
    OR GVL_COMMAND_SHADOW.G_Lock_2_Open
    OR GVL_COMMAND_SHADOW.G_Lock_2_Close
    OR GVL_COMMAND_SHADOW.G_Gate_Open
    OR GVL_COMMAND_SHADOW.G_Wicket_Open
    OR GVL_ACCESS_RUNTIME.G_Any_Pulse_Active;

GVL_DOMAIN_EXECUTION_POLICY.Access_Periodic_Run :=
    (NOT GVL_DOMAIN_EXECUTION_POLICY.Access_Critical_Run)
    AND (
        GVL_DOMAIN_EXECUTION_POLICY.G_Security_Context_Active
        OR GVL_DOMAIN_EXECUTION_POLICY.G_Away_Context_Active
    );

GVL_DOMAIN_EXECUTION_POLICY.Access_Idle_By_Design :=
    NOT GVL_DOMAIN_EXECUTION_POLICY.Access_Critical_Run
    AND NOT GVL_DOMAIN_EXECUTION_POLICY.Access_Periodic_Run;

IF GVL_DOMAIN_EXECUTION_POLICY.Access_Critical_Run THEN
    GVL_DOMAIN_EXECUTION_POLICY.Access_Mode := 2;
ELSIF GVL_DOMAIN_EXECUTION_POLICY.Access_Periodic_Run THEN
    GVL_DOMAIN_EXECUTION_POLICY.Access_Mode := 1;
ELSE
    GVL_DOMAIN_EXECUTION_POLICY.Access_Mode := 0;
END_IF;

GVL_DOMAIN_EXECUTION_POLICY.Lighting_Critical_Run :=
    (GVL_SAFETY_SHUTDOWN.G_Safety_Mode = FIRE)
    OR GVL_STATE.G_Evacuation_Lighting_Active
    OR GVL_LIGHTING_RUNTIME.G_Emergency_Override_Active
    OR GVL_LIGHTING_RUNTIME.G_Any_Light_Active
    OR GVL_LIGHTING_RUNTIME.G_Any_Blind_Not_Safe_Open
    OR GVL_LIGHTING_RUNTIME.G_Any_Socket_Active
    OR GVL_ALARM.G_Security_Alarm;

GVL_DOMAIN_EXECUTION_POLICY.Lighting_Periodic_Run :=
    (NOT GVL_DOMAIN_EXECUTION_POLICY.Lighting_Critical_Run)
    AND (
        GVL_DOMAIN_EXECUTION_POLICY.G_Security_Context_Active
        OR GVL_DOMAIN_EXECUTION_POLICY.G_Away_Context_Active
        OR GVL_DOMAIN_EXECUTION_POLICY.G_Presence_Context_Active
    );

GVL_DOMAIN_EXECUTION_POLICY.Lighting_Idle_By_Design :=
    NOT GVL_DOMAIN_EXECUTION_POLICY.Lighting_Critical_Run
    AND NOT GVL_DOMAIN_EXECUTION_POLICY.Lighting_Periodic_Run;

IF GVL_DOMAIN_EXECUTION_POLICY.Lighting_Critical_Run THEN
    GVL_DOMAIN_EXECUTION_POLICY.Lighting_Mode := 2;
ELSIF GVL_DOMAIN_EXECUTION_POLICY.Lighting_Periodic_Run THEN
    GVL_DOMAIN_EXECUTION_POLICY.Lighting_Mode := 1;
ELSE
    GVL_DOMAIN_EXECUTION_POLICY.Lighting_Mode := 0;
END_IF;

GVL_DOMAIN_EXECUTION_POLICY.Water_Critical_Run :=
    (GVL_SAFETY_SHUTDOWN.G_Safety_Mode = WATER_LEAK)
    OR (GVL_SAFETY_SHUTDOWN.G_Safety_Mode = GLOBAL_STOP)
    OR GVL_COMMAND_SHADOW.G_Water_Block
    OR GVL_COMMAND_SHADOW.G_Water_Emergency_Stop
    OR GVL_COMMAND_SHADOW.G_Close_Valve_35
    OR GVL_COMMAND_SHADOW.G_Close_Valve_36
    OR GVL_WATER_DOMAIN_STATUS.G_Recovery_Requested
    OR GVL_WATER_DOMAIN_STATUS.G_Global_Path_Active
    OR GVL_WATER_DOMAIN_STATUS.G_Output_35_Active
    OR GVL_WATER_DOMAIN_STATUS.G_Output_36_Active
    OR GVL_WATER_DOMAIN_STATUS.G_Any_Zone_Active;

GVL_DOMAIN_EXECUTION_POLICY.Water_Periodic_Run :=
    (NOT GVL_DOMAIN_EXECUTION_POLICY.Water_Critical_Run)
    AND (
        GVL_DOMAIN_EXECUTION_POLICY.G_Security_Context_Active
        OR GVL_DOMAIN_EXECUTION_POLICY.G_Away_Context_Active
    );

GVL_DOMAIN_EXECUTION_POLICY.Water_Idle_By_Design :=
    NOT GVL_DOMAIN_EXECUTION_POLICY.Water_Critical_Run
    AND NOT GVL_DOMAIN_EXECUTION_POLICY.Water_Periodic_Run;

IF GVL_DOMAIN_EXECUTION_POLICY.Water_Critical_Run THEN
    GVL_DOMAIN_EXECUTION_POLICY.Water_Mode := 2;
ELSIF GVL_DOMAIN_EXECUTION_POLICY.Water_Periodic_Run THEN
    GVL_DOMAIN_EXECUTION_POLICY.Water_Mode := 1;
ELSE
    GVL_DOMAIN_EXECUTION_POLICY.Water_Mode := 0;
END_IF;

L_Heating_Output_Active :=
    GVL_HEATING_OUTPUT.DO_DHW_Heating_Pump
    OR GVL_HEATING_OUTPUT.DO_DHW_Circ_Pump
    OR GVL_HEATING_OUTPUT.DO_Backup_Circulation_Pump
    OR GVL_HEATING_OUTPUT.DO_Electric_Heater_Enable;

FOR L_i := 1 TO GVL_CONSTANTS.C_MAX_HEATING_CIRCUITS DO
    L_Heating_Output_Active :=
        L_Heating_Output_Active
        OR GVL_HEATING_OUTPUT.DO_Zone_Valves[L_i];
END_FOR;

FOR L_i := 1 TO GVL_CONSTANTS.C_MAX_MANIFOLDS DO
    L_Heating_Output_Active :=
        L_Heating_Output_Active
        OR GVL_HEATING_OUTPUT.DO_Manifold_Pumps[L_i]
        OR (GVL_HEATING_OUTPUT.AO_Manifold_Valves[L_i] > 0);
END_FOR;

GVL_DOMAIN_EXECUTION_POLICY.Heating_Critical_Run :=
    (GVL_SAFETY_SHUTDOWN.G_Safety_Mode = GAS)
    OR (GVL_SAFETY_SHUTDOWN.G_Safety_Mode = GLOBAL_STOP)
    OR GVL_COMMAND_SHADOW.G_Heating_Block
    OR GVL_COMMAND_SHADOW.G_Heating_Emergency_Stop
    OR GVL_COMMAND_SHADOW.G_Heating_Gas_Safety_Stop
    OR GVL_STATE.G_Safety_Gas_Latched
    OR GVL_STATE.G_Safety_Freeze_Risk
    OR L_Heating_Output_Active;

GVL_DOMAIN_EXECUTION_POLICY.Heating_Periodic_Run :=
    (NOT GVL_DOMAIN_EXECUTION_POLICY.Heating_Critical_Run)
    AND (
        GVL_STATUS.G_Current_Scenario = SCENARIO_MORNING
        OR GVL_STATUS.G_Current_Scenario = SCENARIO_EVENING
        OR GVL_STATUS.G_Current_Scenario = SCENARIO_SLEEP
        OR GVL_STATUS.G_Current_Scenario = SCENARIO_PRESENCE
        OR GVL_INPUT.IN_Preheat_Request
        OR GVL_INPUT.IN_Freeze_Request
    );

GVL_DOMAIN_EXECUTION_POLICY.Heating_Idle_By_Design :=
    NOT GVL_DOMAIN_EXECUTION_POLICY.Heating_Critical_Run
    AND NOT GVL_DOMAIN_EXECUTION_POLICY.Heating_Periodic_Run;

IF GVL_DOMAIN_EXECUTION_POLICY.Heating_Critical_Run THEN
    GVL_DOMAIN_EXECUTION_POLICY.Heating_Mode := 2;
ELSIF GVL_DOMAIN_EXECUTION_POLICY.Heating_Periodic_Run THEN
    GVL_DOMAIN_EXECUTION_POLICY.Heating_Mode := 1;
ELSE
    GVL_DOMAIN_EXECUTION_POLICY.Heating_Mode := 0;
END_IF;

L_Vent_Output_Active := GVL_VENT_OUTPUT.DO_Vent_Enable;

FOR L_i := 1 TO GVL_CONSTANTS.C_MAX_SUPPLY_FANS DO
    L_Vent_Output_Active :=
        L_Vent_Output_Active
        OR (GVL_VENT_OUTPUT.AO_Supply_Fans[L_i] > 0);
END_FOR;

FOR L_i := 1 TO GVL_CONSTANTS.C_MAX_EXHAUST_FANS DO
    L_Vent_Output_Active :=
        L_Vent_Output_Active
        OR (GVL_VENT_OUTPUT.AO_Exhaust_Fans[L_i] > 0);
END_FOR;

GVL_DOMAIN_EXECUTION_POLICY.Vent_Critical_Run :=
    (GVL_SAFETY_SHUTDOWN.G_Safety_Mode = FIRE)
    OR (GVL_SAFETY_SHUTDOWN.G_Safety_Mode = GAS)
    OR (GVL_SAFETY_SHUTDOWN.G_Safety_Mode = GLOBAL_STOP)
    OR GVL_COMMAND_SHADOW.G_Vent_Stop
    OR GVL_COMMAND_SHADOW.G_Vent_Block
    OR GVL_COMMAND_SHADOW.G_Vent_PV3_Boost
    OR GVL_COMMAND_SHADOW.G_Exhaust_100_Req
    OR GVL_COMMAND_SHADOW.G_Vent_Smoke_Exhaust
    OR L_Vent_Output_Active;

GVL_DOMAIN_EXECUTION_POLICY.Vent_Periodic_Run :=
    (NOT GVL_DOMAIN_EXECUTION_POLICY.Vent_Critical_Run)
    AND (
        GVL_DOMAIN_EXECUTION_POLICY.G_Presence_Context_Active
        OR GVL_DOMAIN_EXECUTION_POLICY.G_Away_Context_Active
        OR GVL_INTENT_BEHAVIOR.I_Request_Ventilation_Boost
    );

GVL_DOMAIN_EXECUTION_POLICY.Vent_Idle_By_Design :=
    NOT GVL_DOMAIN_EXECUTION_POLICY.Vent_Critical_Run
    AND NOT GVL_DOMAIN_EXECUTION_POLICY.Vent_Periodic_Run;

IF GVL_DOMAIN_EXECUTION_POLICY.Vent_Critical_Run THEN
    GVL_DOMAIN_EXECUTION_POLICY.Vent_Mode := 2;
ELSIF GVL_DOMAIN_EXECUTION_POLICY.Vent_Periodic_Run THEN
    GVL_DOMAIN_EXECUTION_POLICY.Vent_Mode := 1;
ELSE
    GVL_DOMAIN_EXECUTION_POLICY.Vent_Mode := 0;
END_IF;

GVL_DOMAIN_EXECUTION_POLICY.Simulation_Context_Active :=
    GVL_SIMULATION.G_Test_Scenario_Active
    OR GVL_SIMULATION.G_Test_Start
    OR GVL_DOMAIN_EXECUTION_POLICY.G_Security_Context_Active
    OR GVL_DOMAIN_EXECUTION_POLICY.G_Away_Context_Active;

GVL_DOMAIN_EXECUTION_POLICY.Simulation_Run_Allowed :=
    GVL_SIMULATION.G_Simulation_Enable
    AND GVL_DOMAIN_EXECUTION_POLICY.Simulation_Context_Active
    AND NOT GVL_FABRIC_LIFECYCLE_REGISTRY.Simulation_Suspension_Recommended;

GVL_DOMAIN_EXECUTION_POLICY.Simulation_Idle_By_Design :=
    NOT GVL_DOMAIN_EXECUTION_POLICY.Simulation_Run_Allowed;

IF GVL_DOMAIN_EXECUTION_POLICY.Simulation_Run_Allowed THEN
    GVL_DOMAIN_EXECUTION_POLICY.Simulation_Mode := 1;
ELSE
    GVL_DOMAIN_EXECUTION_POLICY.Simulation_Mode := 0;
END_IF;

GVL_DOMAIN_EXECUTION_POLICY.Any_Critical_Run :=
    GVL_DOMAIN_EXECUTION_POLICY.Access_Critical_Run
    OR GVL_DOMAIN_EXECUTION_POLICY.Lighting_Critical_Run
    OR GVL_DOMAIN_EXECUTION_POLICY.Water_Critical_Run
    OR GVL_DOMAIN_EXECUTION_POLICY.Heating_Critical_Run
    OR GVL_DOMAIN_EXECUTION_POLICY.Vent_Critical_Run;

GVL_DOMAIN_EXECUTION_POLICY.Any_Periodic_Run :=
    GVL_DOMAIN_EXECUTION_POLICY.Access_Periodic_Run
    OR GVL_DOMAIN_EXECUTION_POLICY.Lighting_Periodic_Run
    OR GVL_DOMAIN_EXECUTION_POLICY.Water_Periodic_Run
    OR GVL_DOMAIN_EXECUTION_POLICY.Heating_Periodic_Run
    OR GVL_DOMAIN_EXECUTION_POLICY.Vent_Periodic_Run;

GVL_DOMAIN_EXECUTION_POLICY.Any_Idle_By_Design :=
    GVL_DOMAIN_EXECUTION_POLICY.Access_Idle_By_Design
    OR GVL_DOMAIN_EXECUTION_POLICY.Lighting_Idle_By_Design
    OR GVL_DOMAIN_EXECUTION_POLICY.Water_Idle_By_Design
    OR GVL_DOMAIN_EXECUTION_POLICY.Heating_Idle_By_Design
    OR GVL_DOMAIN_EXECUTION_POLICY.Vent_Idle_By_Design
    OR GVL_DOMAIN_EXECUTION_POLICY.Simulation_Idle_By_Design;

IF GVL_DOMAIN_EXECUTION_POLICY.Any_Critical_Run THEN
    GVL_DOMAIN_EXECUTION_POLICY.Status_Code := 2;
    GVL_DOMAIN_EXECUTION_POLICY.Status_Text := 'Domain execution policy critical activity present';
ELSIF GVL_DOMAIN_EXECUTION_POLICY.Any_Periodic_Run THEN
    GVL_DOMAIN_EXECUTION_POLICY.Status_Code := 1;
    GVL_DOMAIN_EXECUTION_POLICY.Status_Text := 'Domain execution policy periodic activity present';
ELSE
    GVL_DOMAIN_EXECUTION_POLICY.Status_Code := 0;
    GVL_DOMAIN_EXECUTION_POLICY.Status_Text := 'Domain execution policy idle by design';
END_IF;

// >>> BULK_SYNC_ANCHOR: PRG_Domain_Execution_Policy <<<
END_PROGRAM

(* ---- PRG_Domain_Execution_Validation.st ---- *)
PROGRAM PRG_Domain_Execution_Validation
// Observational validation for policy-gated domain execution.
// Detects stale-output risks when a domain is classified idle.
VAR
    L_i : INT;
    L_Access_Output_Active : BOOL;
    L_Lighting_Output_Active : BOOL;
    L_Water_Output_Active : BOOL;
    L_Heating_Output_Active : BOOL;
    L_Vent_Output_Active : BOOL;
END_VAR

GVL_DOMAIN_EXECUTION_VALIDATION.G_Last_Update_MS := GVL_TIME_SERVICE.G_Now_MS;
GVL_DOMAIN_EXECUTION_VALIDATION.G_Validation_Executed := TRUE;
GVL_DOMAIN_EXECUTION_VALIDATION.G_Validation_Valid := TRUE;

L_Access_Output_Active :=
    GVL_ACCESS_OUTPUT.DO_Lock_1_Open
    OR GVL_ACCESS_OUTPUT.DO_Lock_1_Close
    OR GVL_ACCESS_OUTPUT.DO_Lock_2_Open
    OR GVL_ACCESS_OUTPUT.DO_Lock_2_Close
    OR GVL_ACCESS_OUTPUT.DO_Gate_Open
    OR GVL_ACCESS_OUTPUT.DO_Wicket_Open;

L_Lighting_Output_Active := FALSE;
FOR L_i := 1 TO GVL_CONSTANTS.C_MAX_LIGHT_ZONES DO
    L_Lighting_Output_Active :=
        L_Lighting_Output_Active
        OR (GVL_LIGHTING_OUTPUT.AO_Lighting_Levels[L_i] > 0);
END_FOR;
FOR L_i := 1 TO GVL_CONSTANTS.C_MAX_BLINDS DO
    L_Lighting_Output_Active :=
        L_Lighting_Output_Active
        OR (GVL_LIGHTING_OUTPUT.AO_Blinds_Positions[L_i] < 1000);
END_FOR;
FOR L_i := 1 TO GVL_CONSTANTS.C_MAX_SOCKETS DO
    L_Lighting_Output_Active :=
        L_Lighting_Output_Active
        OR GVL_LIGHTING_OUTPUT.DO_Sockets[L_i];
END_FOR;

// Water close outputs are fail-safe holds, not stale activity by themselves.
// Zone enable is the only water output treated as stale when policy says idle.
L_Water_Output_Active := FALSE;
FOR L_i := 1 TO GVL_CONSTANTS.C_MAX_WATER_ZONES DO
    L_Water_Output_Active :=
        L_Water_Output_Active
        OR GVL_WATER_OUTPUT.DO_Water_Zone_Enable[L_i];
END_FOR;

L_Heating_Output_Active :=
    GVL_HEATING_OUTPUT.DO_DHW_Heating_Pump
    OR GVL_HEATING_OUTPUT.DO_DHW_Circ_Pump
    OR GVL_HEATING_OUTPUT.DO_Backup_Circulation_Pump
    OR GVL_HEATING_OUTPUT.DO_Electric_Heater_Enable;
FOR L_i := 1 TO GVL_CONSTANTS.C_MAX_HEATING_CIRCUITS DO
    L_Heating_Output_Active :=
        L_Heating_Output_Active
        OR GVL_HEATING_OUTPUT.DO_Zone_Valves[L_i];
END_FOR;
FOR L_i := 1 TO GVL_CONSTANTS.C_MAX_MANIFOLDS DO
    L_Heating_Output_Active :=
        L_Heating_Output_Active
        OR GVL_HEATING_OUTPUT.DO_Manifold_Pumps[L_i]
        OR (GVL_HEATING_OUTPUT.AO_Manifold_Valves[L_i] > 0);
END_FOR;

L_Vent_Output_Active := GVL_VENT_OUTPUT.DO_Vent_Enable;
FOR L_i := 1 TO GVL_CONSTANTS.C_MAX_SUPPLY_FANS DO
    L_Vent_Output_Active :=
        L_Vent_Output_Active
        OR (GVL_VENT_OUTPUT.AO_Supply_Fans[L_i] > 0);
END_FOR;
FOR L_i := 1 TO GVL_CONSTANTS.C_MAX_EXHAUST_FANS DO
    L_Vent_Output_Active :=
        L_Vent_Output_Active
        OR (GVL_VENT_OUTPUT.AO_Exhaust_Fans[L_i] > 0);
END_FOR;

GVL_DOMAIN_EXECUTION_VALIDATION.Access_Stale_Output_Risk :=
    GVL_DOMAIN_EXECUTION_POLICY.Access_Idle_By_Design AND L_Access_Output_Active;

GVL_DOMAIN_EXECUTION_VALIDATION.Lighting_Stale_Output_Risk :=
    GVL_DOMAIN_EXECUTION_POLICY.Lighting_Idle_By_Design AND L_Lighting_Output_Active;

GVL_DOMAIN_EXECUTION_VALIDATION.Water_Stale_Output_Risk :=
    GVL_DOMAIN_EXECUTION_POLICY.Water_Idle_By_Design AND L_Water_Output_Active;

GVL_DOMAIN_EXECUTION_VALIDATION.Heating_Stale_Output_Risk :=
    GVL_DOMAIN_EXECUTION_POLICY.Heating_Idle_By_Design AND L_Heating_Output_Active;

GVL_DOMAIN_EXECUTION_VALIDATION.Vent_Stale_Output_Risk :=
    GVL_DOMAIN_EXECUTION_POLICY.Vent_Idle_By_Design AND L_Vent_Output_Active;

GVL_DOMAIN_EXECUTION_VALIDATION.Any_Stale_Output_Risk :=
    GVL_DOMAIN_EXECUTION_VALIDATION.Access_Stale_Output_Risk
    OR GVL_DOMAIN_EXECUTION_VALIDATION.Lighting_Stale_Output_Risk
    OR GVL_DOMAIN_EXECUTION_VALIDATION.Water_Stale_Output_Risk
    OR GVL_DOMAIN_EXECUTION_VALIDATION.Heating_Stale_Output_Risk
    OR GVL_DOMAIN_EXECUTION_VALIDATION.Vent_Stale_Output_Risk;

GVL_DOMAIN_EXECUTION_VALIDATION.Any_Policy_Mismatch :=
    GVL_DOMAIN_EXECUTION_VALIDATION.Any_Stale_Output_Risk;

IF GVL_DOMAIN_EXECUTION_VALIDATION.Any_Stale_Output_Risk THEN
    GVL_DOMAIN_EXECUTION_VALIDATION.G_Validation_Valid := FALSE;
    GVL_DOMAIN_EXECUTION_VALIDATION.Status_Code := 1;
    GVL_DOMAIN_EXECUTION_VALIDATION.Status_Text := 'Domain execution validation detected stale output risk';
ELSE
    GVL_DOMAIN_EXECUTION_VALIDATION.Status_Code := 0;
    GVL_DOMAIN_EXECUTION_VALIDATION.Status_Text := 'Domain execution validation nominal';
END_IF;

// >>> BULK_SYNC_ANCHOR: PRG_Domain_Execution_Validation <<<
END_PROGRAM

(* ---- PRG_Energy_Resurrection_Boundary_Governor.st ---- *)
PROGRAM PRG_Energy_Resurrection_Boundary_Governor
IF GVL_POWER_DOMAIN_SEGMENTATION_FABRIC.Power_Domain_Segmentation_Granted
AND NOT GVL_ENERGY_RESURRECTION_BOUNDARY_FABRIC.Unsafe_Energy_Resurrection_Detected
AND NOT GVL_ENERGY_RESURRECTION_BOUNDARY_FABRIC.CrossDomain_Energy_Recovery_Race
AND NOT GVL_ENERGY_RESURRECTION_BOUNDARY_FABRIC.Energy_Recovery_Fork_Detected THEN

    GVL_ENERGY_RESURRECTION_BOUNDARY_FABRIC.Energy_Resurrection_Boundary_Valid := TRUE;
    GVL_ENERGY_RESURRECTION_BOUNDARY_FABRIC.Energy_Resurrection_Boundary_Granted := TRUE;
    GVL_ENERGY_RESURRECTION_BOUNDARY_FABRIC.Energy_Resurrection_Causality_Valid := TRUE;
    GVL_ENERGY_RESURRECTION_BOUNDARY_FABRIC.Energy_Authority_Recovery_Bounded := TRUE;
    GVL_ENERGY_RESURRECTION_BOUNDARY_FABRIC.CrossDomain_Energy_Recovery_Stable := TRUE;
END_IF;
END_PROGRAM

(* ---- PRG_Explainability.st ---- *)
PROGRAM PRG_Explainability
VAR
    L_Mode : E_Safety_Mode;
    L_Recovery : E_Recovery_Phase;
    L_Command : STRING(120);
    L_Heating : STRING(255);
    L_Output : STRING(120);
END_VAR

L_Mode := GVL_SAFETY_SHUTDOWN.G_Safety_Mode;
L_Recovery := GVL_SAFETY_RECOVERY.G_Recovery_Phase;

GVL_EXPLAINABILITY.G_Last_Safety_Mode := L_Mode;
GVL_EXPLAINABILITY.G_Last_Recovery_Phase := L_Recovery;
GVL_EXPLAINABILITY.G_Last_Update_MS := GVL_TIME_SERVICE.G_Now_MS;

CASE L_Mode OF
    FIRE: GVL_EXPLAINABILITY.G_Reason_Chain_Safety := 'FIRE';
    GAS: GVL_EXPLAINABILITY.G_Reason_Chain_Safety := 'GAS';
    WATER_LEAK: GVL_EXPLAINABILITY.G_Reason_Chain_Safety := 'WATER';
    GLOBAL_STOP: GVL_EXPLAINABILITY.G_Reason_Chain_Safety := 'GLOBAL_STOP';
    ELSE
        IF GVL_SAFETY_RECOVERY.G_Recovery_Active OR (GVL_SAFETY_RECOVERY.G_Recovery_Phase <> IDLE) THEN
            GVL_EXPLAINABILITY.G_Reason_Chain_Safety := 'RECOVERY';
        ELSE
            GVL_EXPLAINABILITY.G_Reason_Chain_Safety := 'NORMAL';
        END_IF;
END_CASE;

GVL_EXPLAINABILITY.G_Reason_Chain_Behavior := GVL_INTENT_BEHAVIOR.I_Reason_Text;

IF GVL_COMMAND_SHADOW.G_Heating_Block THEN
    L_Command := 'Heating Blocked';
ELSIF GVL_COMMAND_SHADOW.G_Vent_Stop THEN
    L_Command := 'Vent Stopped';
ELSIF GVL_COMMAND_SHADOW.G_Water_Block THEN
    L_Command := 'Water Blocked';
ELSE
    L_Command := 'Command OK';
END_IF;
GVL_EXPLAINABILITY.G_Reason_Chain_Command := L_Command;

IF GVL_STATE.G_Heating_RootCause <> E_Heating_RootCause.RC_NONE THEN
    L_Heating := GVL_STATE.G_Heating_Confidence_Reason_Text;
ELSIF GVL_STATE.G_Heating_Cascade_Degraded THEN
    L_Heating := 'Heating cascade degraded';
ELSE
    L_Heating := 'Heating OK';
END_IF;
GVL_EXPLAINABILITY.G_Heating_Why_Blocked := L_Heating;

IF GVL_COMMAND_VERIFY.PreOutput_Block_IO THEN
    L_Output := 'Outputs held by PreOutput barrier';
ELSIF GVL_SAFETY_RECOVERY.G_Recovery_Phase <> IDLE THEN
    L_Output := 'Outputs held during recovery';
ELSIF GVL_RUNTIME_IO_VALIDATION.Any_IO_Invalid THEN
    L_Output := 'Outputs applied with IO validation mismatch';
ELSE
    L_Output := 'Outputs Applied';
END_IF;
GVL_EXPLAINABILITY.G_Reason_Chain_Output := L_Output;

GVL_EXPLAINABILITY.G_Reason_Chain_Full := CONCAT(
    CONCAT(
        CONCAT(
            GVL_EXPLAINABILITY.G_Reason_Chain_Safety,
            ' -> '
        ),
        CONCAT(
            GVL_EXPLAINABILITY.G_Reason_Chain_Behavior,
            ' -> '
        )
    ),
    CONCAT(
        CONCAT(
            GVL_EXPLAINABILITY.G_Reason_Chain_Command,
            ' -> '
        ),
        CONCAT(
            L_Heating,
            CONCAT(' -> ', L_Output)
        )
    )
);

GVL_EXPLAINABILITY.G_Behavior_Why_Active := GVL_INTENT_BEHAVIOR.I_Reason_Text;

END_PROGRAM

(* ---- PRG_File_Archive_Manager.st ---- *)
PROGRAM PRG_File_Archive_Manager
// ==============================================================================
// FILE ARCHIVE MANAGER — deterministic runtime surface for future CSV/file export.
// ==============================================================================
// No direct file, USB or gateway write is implemented here. This program only
// consumes one-shot archive requests, validates the configured target surface and
// publishes a deterministic status/error until concrete CODESYS file libraries
// and port-specific paths are selected.
// ==============================================================================
VAR
    L_Request_Active : BOOL;
    L_Target_Available : BOOL;
END_VAR

// Daily automatic configuration backup scheduler. It publishes the same
// one-shot request as HMI/gateway paths and never writes files directly.
IF GVL_FILE_ARCHIVE.G_Auto_Config_Backup_Enabled THEN
    IF (GVL_TIME_SERVICE.G_Day_Of_Week >= 1) AND
       (GVL_TIME_SERVICE.G_Day_Of_Week <= 7) AND
       (GVL_TIME_SERVICE.G_Time_Of_Day_MS >= GVL_FILE_ARCHIVE.G_Auto_Config_Backup_Time_Of_Day_MS) THEN
        IF GVL_FILE_ARCHIVE.G_Auto_Config_Backup_Last_Day_Of_Week <> GVL_TIME_SERVICE.G_Day_Of_Week THEN
            GVL_FILE_ARCHIVE.G_Write_Config_Backup_Request := TRUE;
            GVL_FILE_ARCHIVE.G_Auto_Config_Backup_Last_Day_Of_Week := GVL_TIME_SERVICE.G_Day_Of_Week;
            GVL_FILE_ARCHIVE.G_Auto_Config_Backup_Last_Request_MS := GVL_TIME_SERVICE.G_Now_MS;
            GVL_FILE_ARCHIVE.G_Auto_Config_Backup_Last_Status_Text := 'Auto config backup request published';
        END_IF;
    END_IF;
END_IF;

L_Request_Active :=
    GVL_FILE_ARCHIVE.G_Write_Event_CSV_Request
    OR GVL_FILE_ARCHIVE.G_Write_Trend_CSV_Request
    OR GVL_FILE_ARCHIVE.G_Write_BlackBox_CSV_Request
    OR GVL_FILE_ARCHIVE.G_Write_Config_Backup_Request;

L_Target_Available := FALSE;
CASE GVL_FILE_ARCHIVE.G_File_Archive_Target_Code OF
    1:
        L_Target_Available := GVL_FILE_ARCHIVE.G_PLC_File_Target_Available;
    2:
        L_Target_Available := GVL_FILE_ARCHIVE.G_USB_Target_Available;
    3:
        L_Target_Available := GVL_FILE_ARCHIVE.G_Gateway_Target_Available;
ELSE
    L_Target_Available := FALSE;
END_CASE;

IF L_Request_Active THEN
    GVL_FILE_ARCHIVE.G_Write_Busy := FALSE;
    GVL_FILE_ARCHIVE.G_Write_Done := FALSE;
    GVL_FILE_ARCHIVE.G_Write_Error := FALSE;
    GVL_FILE_ARCHIVE.G_Last_Error_Code := 0;
    GVL_FILE_ARCHIVE.G_Last_Status_Text := '';
    GVL_FILE_ARCHIVE.G_Last_Write_MS := GVL_TIME_SERVICE.G_Now_MS;

    IF NOT GVL_FILE_ARCHIVE.G_Archive_Interface_Enabled THEN
        GVL_FILE_ARCHIVE.G_Write_Error := TRUE;
        GVL_FILE_ARCHIVE.G_Last_Error_Code := 16#A001;
        GVL_FILE_ARCHIVE.G_Last_Status_Text := 'Archive interface disabled';
    ELSIF NOT GVL_FILE_ARCHIVE.G_CSV_Write_Enabled THEN
        GVL_FILE_ARCHIVE.G_Write_Error := TRUE;
        GVL_FILE_ARCHIVE.G_Last_Error_Code := 16#A002;
        GVL_FILE_ARCHIVE.G_Last_Status_Text := 'CSV archive disabled';
    ELSIF GVL_FILE_ARCHIVE.G_File_Archive_Target_Code = 0 THEN
        GVL_FILE_ARCHIVE.G_Write_Error := TRUE;
        GVL_FILE_ARCHIVE.G_Last_Error_Code := 16#A003;
        GVL_FILE_ARCHIVE.G_Last_Status_Text := 'No archive target selected';
    ELSIF NOT L_Target_Available THEN
        GVL_FILE_ARCHIVE.G_Write_Error := TRUE;
        GVL_FILE_ARCHIVE.G_Last_Error_Code := 16#A004;
        GVL_FILE_ARCHIVE.G_Last_Status_Text := 'Selected archive target unavailable';
    ELSE
        GVL_FILE_ARCHIVE.G_Write_Error := TRUE;
        GVL_FILE_ARCHIVE.G_Last_Error_Code := 16#A005;
        GVL_FILE_ARCHIVE.G_Last_Status_Text := 'Archive backend not connected';
    END_IF;

    // One-shot requests are consumed regardless of the result so HMI/gateway
    // callers receive a stable status instead of repeatedly retriggering.
    GVL_FILE_ARCHIVE.G_Write_Event_CSV_Request := FALSE;
    GVL_FILE_ARCHIVE.G_Write_Trend_CSV_Request := FALSE;
    GVL_FILE_ARCHIVE.G_Write_BlackBox_CSV_Request := FALSE;
    GVL_FILE_ARCHIVE.G_Write_Config_Backup_Request := FALSE;
END_IF;

// >>> BULK_SYNC_ANCHOR: PRG_File_Archive_Manager <<<
END_PROGRAM
